Universal Robots PolyScope program: 958_16_OCT_2021_IZQ.urp

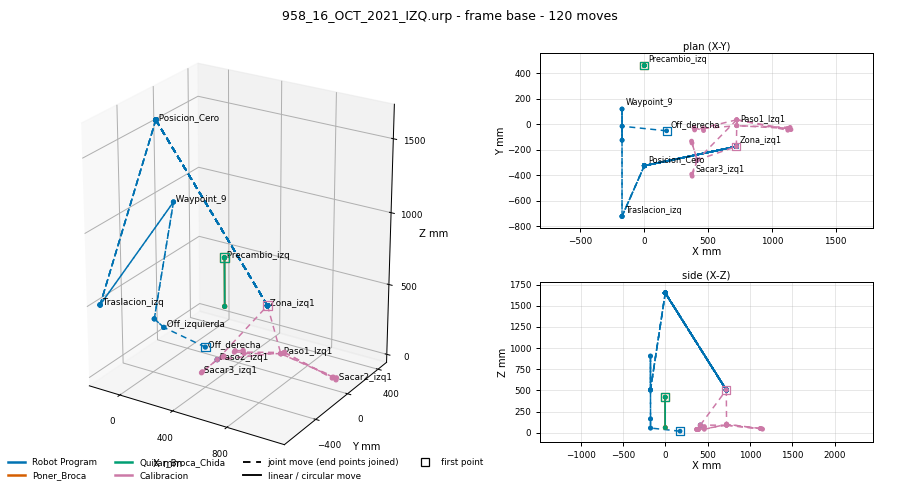
[picture p0: tool path of 958_16_OCT_2021_IZQ.urp in frame base, 120 of 216 moves have a stored position in this frame; points joined in program order, loops and branches not executed]
Program 958_16_OCT_2021_IZQ (installation=instalacion_derecha_10_MAR_21 directory=/programs/FAI3 createdIn=5.6.0.90886 lastSavedIn=5.11.1.108318 robotSerialNumber=20195001785)
Calibrated DH parameters: a=[0.000107, -0.568984, -0.552934, -0.00001, -0.000063, 0]; d=[0.180718, -257.998067, 200.685024, 57.48776, 0.119923, 0.115353]; alpha=[1.571119, 0.000876, -0.002498, 1.571178, -1.570523, 0]; deltaTheta=[0, -0.378191, 0.631587, -0.253396, 0, 0]
Robot Program (runOnlyOnce=false)
  SuppressedNode
    Folder Pruebas_cambiador
      MoveJ speed 60 deg/s, acceleration 80 deg/s^2 (useActiveTCP=true) feature=Base
        Waypoint Precambio_izq: TCP in base x=0.343 y=460.224 z=419.989 mm, rx=0.2109 ry=3.1246 rz=-0.0222 rad; joints [-122.778, -120.749, 120.698, 0.478, 59.722, -0.747] deg; TCP offset x=0.151 y=-167.165 z=35.088 mm, rx=1.5784 ry=-0.0729 rz=0.0687 rad
      Loop Forever
        Call Poner_Broca
        Call Quitar_Broca_Chida
  SuppressedNode
    'Programa'
  Set DigitalOutput pin=salida0; digitalValue=1
  broca := 1645
  Script: textmsg("----------DAS-----------")
  Set ExpressionOutput pin=mensaje_mw10; expression=15
  Wait DigitalInput pin=Continuar_M30; digitalValue=1
  Wait Sleep waitTime=1
  If Lado_Correr≟1
    Folder Arranque
      MoveJ speed 30 deg/s, acceleration 50 deg/s^2 (useActiveTCP=true) feature=Base
        Waypoint Off_derecha: TCP in base x=175.169 y=-51.554 z=18.125 mm, rx=-2.0046 ry=0.0915 rz=0.0578 rad; joints [90.003, -90, 154.529, 0, 89.998, -0.004] deg
        Waypoint Off_izquierda: TCP in base x=-173.642 y=-15.442 z=55.621 mm, rx=-1.8394 ry=0.083 rz=0.0614 rad; joints [-89.997, -89.996, -154.003, -190.002, -89.995, 0.005] deg
      Set DigitalOutput pin=postrnas_m187; digitalValue=1
      Wait Sleep waitTime=1
      Set DigitalOutput pin=Home_M20; digitalValue=1
      Wait Sleep waitTime=1
      Set DigitalOutput pin=postrnas_m187; digitalValue=0
      Set DigitalOutput pin=Home_M20; digitalValue=0
      Set ExpressionOutput pin=mensaje_mw10; expression=20
      Wait DigitalInput pin=Continuar_M30; digitalValue=1
      Wait Sleep waitTime=1
    Folder Traslacion
      Set ExpressionOutput pin=mensaje_mw10; expression=25
      Wait DigitalInput pin=Continuar_M30; digitalValue=1
      Wait Sleep waitTime=1
      MoveJ speed 60 deg/s, acceleration 80 deg/s^2 (useActiveTCP=true) feature=Base
        Waypoint Waypoint_8: TCP in base x=-173.7 y=-124.883 z=163.166 mm, rx=3.1302 ry=-0.1403 rz=0.0027 rad; joints [-90.002, -15, -153.998, -189.998, -89.998, -0.004] deg
        Waypoint Waypoint_9: TCP in base x=-174.329 y=119.284 z=905.669 mm, rx=2.0147 ry=-0.0908 rz=0.0576 rad; joints [-90.002, -15.002, -90.002, -189.996, -89.997, -0.004] deg
        Waypoint Traslacion_izq: TCP in base x=-174.237 y=-721.63 z=505.386 mm, rx=-3.1292 ry=0.1412 rz=-0.0002 rad; joints [-90, -90.001, -90.002, -180, -90.003, -0.001] deg
      Set ExpressionOutput pin=mensaje_mw10; expression=30
      Wait DigitalInput pin=Continuar_M30; digitalValue=1
      Wait Sleep waitTime=1
      Set DigitalOutput pin=postrnas_m187; digitalValue=1
      Wait Sleep waitTime=1
      Set DigitalOutput pin=pos1_izq_m22; digitalValue=1
      Wait Sleep waitTime=2
      Set DigitalOutput pin=pos1_izq_m22; digitalValue=0
      Set DigitalOutput pin=postrnas_m187; digitalValue=0
      Wait Sleep waitTime=5
      Set ExpressionOutput pin=mensaje_mw10; expression=35
      Wait DigitalInput pin=Continuar_M30; digitalValue=1
      Wait Sleep waitTime=1
    Folder Brocas
      Set DigitalOutput pin=carrusel_home; digitalValue=1
      Wait Sleep waitTime=1
      Set DigitalOutput pin=carrusel_home; digitalValue=0
      Set ExpressionOutput pin=mensaje_mw10; expression=40
      Wait DigitalInput pin=Continuar_M30; digitalValue=1
      Wait Sleep waitTime=1
      Set DigitalOutput pin=carrusel_home; digitalValue=1
      Wait Sleep waitTime=1
      Set DigitalOutput pin=carrusel_home; digitalValue=0
      Set ExpressionOutput pin=mensaje_mw10; expression=45
      Wait DigitalInput pin=Continuar_M30; digitalValue=1
      Wait Sleep waitTime=1
      Call Poner_Broca
    Folder Offsets factor
      SuppressedNode
        broca := 1645
      L1B1x := ((0.09523476)/(0.09525))*(0.09523476)
      L1B1y := ((-0.01278382)/(-0.0127))*(-0.01278382)
      L1B2x := ((0.75575414)/(0.75565))*(0.75575414)
      L1B2y := ((-0.01279398)/(-0.0127))*(-0.01279398)
      L2B1x := ((0.09675299)/(0.09525))*(0.09675299)
      L2B1y := ((0.3937)/(0.3937))*(0.3937)
      L2B2x := ((0.757306777)/(0.75565))*(0.757306777)
      L2B2y := ((0.393684081)/(0.3937))*(0.393684081)
    Folder Calibracion
      Set ExpressionOutput pin=mensaje_mw10; expression=50
      Wait DigitalInput pin=Continuar_M30; digitalValue=1
      Wait Sleep waitTime=1
      MoveJ speed 60 deg/s, acceleration 80 deg/s^2 (useActiveTCP=true) feature=Base
        Waypoint Posicion_Cero: TCP in base x=0.551 y=-324.742 z=1651.532 mm, rx=-0.0041 ry=-0.0154 rz=-3.05 rad; joints [-0.003, -90.003, 0.004, -89.999, -0.001, 0] deg
        Waypoint Zona_izq1: TCP in base x=721.637 y=-174.262 z=505.425 mm, rx=2.3235 ry=2.1144 rz=0.0001 rad; joints [0.067, -89.734, -90.405, -179.332, -89.71, -0.034] deg
      broca := 1645
      Set ExpressionOutput pin=mensaje_mw10; expression=125
      Wait DigitalInput pin=Continuar_M30; digitalValue=1
      Wait Sleep waitTime=1
      Set ExpressionOutput pin=mensaje_mw10; expression=130
      Wait DigitalInput pin=Continuar_M30; digitalValue=1
      Wait Sleep waitTime=1
      Call Calibracion
    Folder GoNoGo
      Set ExpressionOutput pin=mensaje_mw10; expression=55
      Wait DigitalInput pin=Continuar_M30; digitalValue=1
      Wait Sleep waitTime=1
      Set ExpressionOutput pin=mensaje_mw10; expression=60
      Wait DigitalInput pin=Continuar_M30; digitalValue=1
      Wait Sleep waitTime=1
      Folder Linea1_Buje1
        Xfin := ((((L1B1x)*(-1)*Xp)-(Xd)-((L1B1y)*(1/m2)))*(-1))*(1)
        Yfin := ((((L1B1y)*(-1)*Yp)-(Yd)+((L1B1x)*(-1)*m1))*(-1))*(1)
        rotaciones := get_actual_tcp_pose()
        var_3 := rotaciones[3]
        var_4 := rotaciones[4]
        var_5 := rotaciones[5]
        If broca≟1645
          PosFinal := p[Xfin-0.00208915,Yfin-0.00208915,0.15,var_3,var_4,var_5]
        ElseIf broca≟1935
          PosFinal := p[Xfin-0.00245745,Yfin-0.00245745,0.15,var_3,var_4,var_5]
        ElseIf broca≟217
          PosFinal := p[Xfin-0.0027559,Yfin-0.0027559,0.15,var_3,var_4,var_5]
        Buje_Final := PosFinal
      MoveJ speed 60 deg/s, acceleration 80 deg/s^2 (useActiveTCP=true) feature=Base
        Waypoint Waypoint (Variable): variable(name=Buje_Final)
      Wait Sleep waitTime=1
      Folder Alturas
        If P1h[2]<P2h[2]
          tcp_chido := get_actual_tcp_pose()
          offset_bajada := p[tcp_chido[0],tcp_chido[1],((alta-0.0095)-(altura/1000)),tcp_chido[3],tcp_chido[4],tcp_chido[5]]
          MoveL speed 15 mm/s, acceleration 30 mm/s^2 (useActiveTCP=true) feature=Base
            Waypoint Waypoint (Variable): variable(name=offset_bajada)
        Else 
          tcp_chido := get_actual_tcp_pose()
          offset_bajada := p[tcp_chido[0],tcp_chido[1],((alta-0.0095)),tcp_chido[3],tcp_chido[4],tcp_chido[5]]
          MoveL speed 15 mm/s, acceleration 30 mm/s^2 (useActiveTCP=true) feature=Base
            Waypoint Waypoint (Variable): variable=offset_bajada
      MoveL speed 15 mm/s, acceleration 30 mm/s^2 (useActiveTCP=true) feature=Base
        Folder Freemove
          Wait Sleep waitTime=2
          Script: freedrive_mode()
          Wait Sleep waitTime=2.5
          Script: end_freedrive_mode()
          var_13 := get_actual_tcp_pose()
          var_13 := p[var_13[0]*1000,var_13[1]*1000,420,420,420,420]
          var_13 := get_actual_tcp_pose()
          var_13 := p[var_13[0],var_13[1],0.1,var_13[3],var_13[4],var_13[5]]
        MoveDirectionNode (selectedDirection=ZPlus)
          Until DISTANCE (allowActions=false deceleration=3 distanceNodeType=STOP) Distance=0.15; motionParameters(blendRadius=0)
      L1B1 := var_13
      Folder Linea1_Buje2
        Xfin := ((((L1B2x)*(-1)*Xp)-(Xd)-((L1B2y)*(1/m2)))*(-1))*(1)
        Yfin := ((((L1B2y)*(-1)*Yp)-(Yd)+((L1B2x)*(-1)*m1))*(-1))*(1)
        rotaciones := get_actual_tcp_pose()
        var_3 := rotaciones[3]
        var_4 := rotaciones[4]
        var_5 := rotaciones[5]
        If broca≟1645
          PosFinal := p[Xfin-0.00208915,Yfin-0.00208915,0.15,var_3,var_4,var_5]
        ElseIf broca≟1935
          PosFinal := p[Xfin-0.00245745,Yfin-0.00245745,0.15,var_3,var_4,var_5]
        ElseIf broca≟217
          PosFinal := p[Xfin-0.0027559,Yfin-0.0027559,0.15,var_3,var_4,var_5]
        Buje_Final := PosFinal
      MoveJ speed 60 deg/s, acceleration 80 deg/s^2 (useActiveTCP=true) feature=Base
        Waypoint Waypoint (Variable): variable=Buje_Final
      Wait Sleep waitTime=1
      Folder Alturas
        If P1h[2]<P2h[2]
          tcp_chido := get_actual_tcp_pose()
          offset_bajada := p[tcp_chido[0],tcp_chido[1],((alta-0.0095)),tcp_chido[3],tcp_chido[4],tcp_chido[5]]
          MoveL speed 15 mm/s, acceleration 30 mm/s^2 (useActiveTCP=true) feature=Base
            Waypoint Waypoint (Variable): variable=offset_bajada
        Else 
          tcp_chido := get_actual_tcp_pose()
          offset_bajada := p[tcp_chido[0],tcp_chido[1],((alta-0.0095)-(altura/1000)),tcp_chido[3],tcp_chido[4],tcp_chido[5]]
          MoveL speed 15 mm/s, acceleration 30 mm/s^2 (useActiveTCP=true) feature=Base
            Waypoint Waypoint (Variable): variable=offset_bajada
      MoveL speed 15 mm/s, acceleration 30 mm/s^2 (useActiveTCP=true) feature=Base
        Folder Freemove
          Wait Sleep waitTime=2
          Script: freedrive_mode()
          Wait Sleep waitTime=2.5
          Script: end_freedrive_mode()
          var_13 := get_actual_tcp_pose()
          var_13 := p[var_13[0]*1000,var_13[1]*1000,420,420,420,420]
          var_13 := get_actual_tcp_pose()
          var_13 := p[var_13[0],var_13[1],0.1,var_13[3],var_13[4],var_13[5]]
        MoveDirectionNode (selectedDirection=ZPlus)
          Until DISTANCE (allowActions=false deceleration=3 distanceNodeType=STOP) Distance=0.15; motionParameters(blendRadius=0)
      L1B2 := var_13
      Folder Linea2_Buje2
        Xfin := ((((L2B2x)*(-1)*Xp)-(Xd)-(L2B2y*(1/m2)))*(-1))*(1)
        Yfin := ((((L2B2y)*(-1)*Yp)-(Yd)+((L2B2x)*(-1)*m1))*(-1))*(1)
        rotaciones := get_actual_tcp_pose()
        var_3 := rotaciones[3]
        var_4 := rotaciones[4]
        var_5 := rotaciones[5]
        If broca≟1645
          PosFinal := p[Xfin-0.00208915,Yfin-0.00208915,0.15,var_3,var_4,var_5]
        ElseIf broca≟1935
          PosFinal := p[Xfin-0.00245745,Yfin-0.00245745,0.15,var_3,var_4,var_5]
        ElseIf broca≟217
          PosFinal := p[Xfin-0.0027559,Yfin-0.0027559,0.15,var_3,var_4,var_5]
        Buje_Final := PosFinal
      MoveJ speed 60 deg/s, acceleration 80 deg/s^2 (useActiveTCP=true) feature=Base
        Waypoint Waypoint (Variable): variable=Buje_Final
      Wait Sleep waitTime=1
      Folder Alturas
        If P1h[2]<P2h[2]
          tcp_chido := get_actual_tcp_pose()
          offset_bajada := p[tcp_chido[0],tcp_chido[1],((alta-0.0095)),tcp_chido[3],tcp_chido[4],tcp_chido[5]]
          MoveL speed 15 mm/s, acceleration 30 mm/s^2 (useActiveTCP=true) feature=Base
            Waypoint Waypoint (Variable): variable=offset_bajada
        Else 
          tcp_chido := get_actual_tcp_pose()
          offset_bajada := p[tcp_chido[0],tcp_chido[1],((alta-0.0095)-(altura/1000)),tcp_chido[3],tcp_chido[4],tcp_chido[5]]
          MoveL speed 15 mm/s, acceleration 30 mm/s^2 (useActiveTCP=true) feature=Base
            Waypoint Waypoint (Variable): variable=offset_bajada
      MoveL speed 15 mm/s, acceleration 30 mm/s^2 (useActiveTCP=true) feature=Base
        Folder Freemove
          Wait Sleep waitTime=2
          Script: freedrive_mode()
          Wait Sleep waitTime=2.5
          Script: end_freedrive_mode()
          var_13 := get_actual_tcp_pose()
          var_13 := p[var_13[0]*1000,var_13[1]*1000,420,420,420,420]
          var_13 := get_actual_tcp_pose()
          var_13 := p[var_13[0],var_13[1],0.1,var_13[3],var_13[4],var_13[5]]
        MoveDirectionNode (selectedDirection=ZPlus)
          Until DISTANCE (allowActions=false deceleration=3 distanceNodeType=STOP) Distance=0.15; motionParameters(blendRadius=0)
      L2B2 := var_13
      Folder Linea2_Buje1
        Xfin := ((((L2B1x)*(-1)*Xp)-(Xd)-((L2B1y)*(1/m2)))*(-1))*(1)
        Yfin := ((((L2B1y)*(-1)*Yp)-(Yd)+((L2B1x)*(-1)*m1))*(-1))*(1)
        rotaciones := get_actual_tcp_pose()
        var_3 := rotaciones[3]
        var_4 := rotaciones[4]
        var_5 := rotaciones[5]
        If broca≟1645
          PosFinal := p[Xfin-0.00208915,Yfin-0.00208915,0.15,var_3,var_4,var_5]
        ElseIf broca≟1935
          PosFinal := p[Xfin-0.00245745,Yfin-0.00245745,0.15,var_3,var_4,var_5]
        ElseIf broca≟217
          PosFinal := p[Xfin-0.0027559,Yfin-0.0027559,0.15,var_3,var_4,var_5]
        Buje_Final := PosFinal
      MoveJ speed 60 deg/s, acceleration 80 deg/s^2 (useActiveTCP=true) feature=Base
        Waypoint Paso2_izq1: TCP in base x=414.118 y=-280.673 z=89.978 mm, rx=-2.3928 ry=-2.0356 rz=0 rad; joints [-18.236, -84.335, -142.099, -133.065, -104.295, 0.11] deg
        Waypoint Waypoint (Variable): variable=Buje_Final
      Wait Sleep waitTime=1
      Folder Alturas
        If P1h[2]<P2h[2]
          tcp_chido := get_actual_tcp_pose()
          offset_bajada := p[tcp_chido[0],tcp_chido[1],((alta-0.0095)-(altura/1000)),tcp_chido[3],tcp_chido[4],tcp_chido[5]]
          MoveL speed 15 mm/s, acceleration 30 mm/s^2 (useActiveTCP=true) feature=Base
            Waypoint Waypoint (Variable): variable=offset_bajada
        Else 
          tcp_chido := get_actual_tcp_pose()
          offset_bajada := p[tcp_chido[0],tcp_chido[1],((alta-0.0095)),tcp_chido[3],tcp_chido[4],tcp_chido[5]]
          MoveL speed 15 mm/s, acceleration 30 mm/s^2 (useActiveTCP=true) feature=Base
            Waypoint Waypoint (Variable): variable=offset_bajada
      MoveL speed 15 mm/s, acceleration 30 mm/s^2 (useActiveTCP=true) feature=Base
        Folder Freemove
          Wait Sleep waitTime=2
          Script: freedrive_mode()
          Wait Sleep waitTime=2.5
          Script: end_freedrive_mode()
          var_13 := get_actual_tcp_pose()
          var_13 := p[var_13[0]*1000,var_13[1]*1000,420,420,420,420]
          var_13 := get_actual_tcp_pose()
          var_13 := p[var_13[0],var_13[1],0.1,var_13[3],var_13[4],var_13[5]]
        MoveDirectionNode (selectedDirection=ZPlus)
          Until DISTANCE (allowActions=false deceleration=3 distanceNodeType=STOP) Distance=0.15; motionParameters(blendRadius=0)
      MoveJ speed 60 deg/s, acceleration 80 deg/s^2 (useActiveTCP=true) feature=Base
        Waypoint Zona_izq1: TCP in base x=721.637 y=-174.262 z=505.425 mm, rx=2.3235 ry=2.1144 rz=0.0001 rad; joints [0.067, -89.734, -90.405, -179.332, -89.71, -0.034] deg
      L2B1 := var_13
    SuppressedNode
      Folder Cancelar barrenado
        MoveJ speed 60 deg/s, acceleration 80 deg/s^2 (useActiveTCP=true) feature=Base
          SuppressedNode
            Waypoint Zona_der1: TCP in base x=-724.618 y=-175.006 z=455.096 mm, rx=2.0346 ry=-2.3862 rz=-0.0105 rad; joints [0.001, -89.997, 90, 0.002, 90.001, 0.002] deg; TCP offset x=0.411 y=-218.298 z=37.994 mm, rx=1.558 ry=-0.1255 rz=0.1212 rad
          Waypoint Zona_izq1: TCP in base x=721.637 y=-174.262 z=505.425 mm, rx=2.3235 ry=2.1144 rz=0.0001 rad; joints [0.067, -89.734, -90.405, -179.332, -89.71, -0.034] deg; TCP offset x=0.151 y=-167.165 z=35.088 mm, rx=1.5784 ry=-0.0729 rz=0.0687 rad
          Waypoint Posicion_Cero: TCP in base x=0.551 y=-324.742 z=1651.532 mm, rx=-0.0041 ry=-0.0154 rz=-3.05 rad; joints [-0.003, -90.003, 0.004, -89.999, -0.001, 0] deg
        Call Quitar_Broca_Chida
        Set ExpressionOutput pin=mensaje_mw10; expression=100
        Wait DigitalInput pin=Continuar_M30; digitalValue=1
        Wait Sleep waitTime=1
        Set ExpressionOutput pin=mensaje_mw10; expression=155
        Wait DigitalInput pin=Continuar_M30; digitalValue=1
        Wait Sleep waitTime=1
    Folder Colocar broca
      Call Quitar_Broca_Chida
      Call Poner_Broca
    Folder Barrenado1
      Set ExpressionOutput pin=mensaje_mw10; expression=65
      Wait DigitalInput pin=Continuar_M30; digitalValue=1
      Wait Sleep waitTime=1
      Set ExpressionOutput pin=mensaje_mw10; expression=150
      Wait Sleep waitTime=1
      Folder Linea 1 a 1645
        broca := 1645
        Folder Buje_inicial
          Buje_Inicial := L1B2
        Folder Buje_final
          Buje_Final := L1B1
        barrenosTotales := 27
        barrenoActual := 1
        Loop While (checkContinuously=false) expression=barrenoActual≤barrenosTotales
          MoveL speed 250 mm/s, acceleration 1200 mm/s^2 (useActiveTCP=true) feature=Base
            bajada_broca := p[0,0,0.006,0,0,0]
            internos := interpolate_pose(Buje_Inicial, Buje_Final, ((barrenoActual)-1)/((barrenosTotales)-1))
            Folder Alturas
              If barrenoActual≟3 or barrenoActual≟5 or barrenoActual≟7 or barrenoActual≟9 or barrenoActual≟11 or barrenoActual≟13 or barrenoActual≟15 or barrenoActual≟17 or barrenoActual≟19 or barrenoActual≟21 or barrenoActual≟23 or barrenoActual≟25 or barrenoActual≟27 or barrenoActual≟1
                Set ExpressionOutput pin=mensaje_mw10; expression=200
                Wait DigitalInput pin=Continuar_M30; digitalValue=1
                Wait Sleep waitTime=1
                Set ExpressionOutput pin=mensaje_mw10; expression=150
                Wait Sleep waitTime=1
              MoveJ speed 60 deg/s, acceleration 80 deg/s^2 (useActiveTCP=true) feature=Base
                Waypoint Waypoint (Variable): variable(name=internos)
              Wait Sleep waitTime=2
              If P1h[2]<P2h[2]
                acomodin := (altura/(barrenosTotales-1))*(barrenoActual-1)
                tcp_chido := get_actual_tcp_pose()
                offset_bajada := p[tcp_chido[0],tcp_chido[1],((alta-0.0095)-(acomodin/1000)),tcp_chido[3],tcp_chido[4],tcp_chido[5]]
                MoveL speed 15 mm/s, acceleration 30 mm/s^2 (useActiveTCP=true) feature=Base
                  Waypoint Waypoint (Variable): variable=offset_bajada
              Else 
                acomodin := (altura/(barrenosTotales-1))*(26-(barrenoActual-1))
                tcp_chido := get_actual_tcp_pose()
                offset_bajada := p[tcp_chido[0],tcp_chido[1],((alta-0.0095)-(acomodin/1000)),tcp_chido[3],tcp_chido[4],tcp_chido[5]]
                MoveL speed 15 mm/s, acceleration 30 mm/s^2 (useActiveTCP=true) feature=Base
                  Waypoint Waypoint (Variable): variable=offset_bajada
            Folder Freemove
              Wait Sleep waitTime=2
              Script: freedrive_mode()
              Wait Sleep waitTime=2.5
              Script: end_freedrive_mode()
            Wait Sleep waitTime=0.3
            Set DigitalOutput pin=config_out[1]; digitalValue=1
            Wait Sleep waitTime=1
            Wait Sleep waitTime=0.3
            Wait Sleep waitTime=0.3
            Wait Sleep waitTime=0.3
            Loop Counting (count=3) loopVariable(name=Loop_4)
              Poses_taladrado := pose_sub(get_actual_tcp_pose(), bajada_broca)
              Waypoint Waypoint (Variable): motionParameters(jointSpeed=1.047198 jointAcceleration=1.396263 cartesianSpeed=0.001 cartesianAcceleration=0.005); variable(name=Poses_taladrado)
              If bajada_broca≟p[0,0,0.018,0,0,0]
                num_barreno := str_cat("Barreno: ",barrenoActual)
                tcp_actual := get_actual_tcp_pose()
                X_actual := str_cat("     X: ",tcp_actual[0])
                Y_actual := str_cat("     Y: ",tcp_actual[1])
                pos_barreno := str_cat(X_actual,Y_actual)
                Script: textmsg(num_barreno,pos_barreno)
              Poses_taladrado := pose_add(get_actual_tcp_pose(), bajada_broca)
              Waypoint Waypoint (Variable): motionParameters(jointSpeed=1.047198 jointAcceleration=1.396263 cartesianSpeed=0.01 cartesianAcceleration=0.01); variable=Poses_taladrado
              bajada_broca := pose_add(bajada_broca, p[0,0,0.006,0,0,0])
            MoveDirectionNode (selectedDirection=ZPlus toolParams=0.03, 0.04)
              Until DISTANCE (allowActions=false deceleration=3 distanceNodeType=STOP) Distance=0.05; motionParameters(blendRadius=0)
            MoveJ speed 60 deg/s, acceleration 80 deg/s^2 (useActiveTCP=true) feature=Base
              Waypoint Waypoint (Variable): variable=internos
            Wait Sleep waitTime=0.3
            Set DigitalOutput pin=config_out[1]; digitalValue=0
            Wait Sleep waitTime=0.3
            If barrenoActual≟13 or barrenoActual≟27
              MoveDirectionNode (selectedDirection=ZPlus toolParams=0.03, 0.04)
                Until DISTANCE (allowActions=false deceleration=3 distanceNodeType=STOP) Distance=0.03; motionParameters(blendRadius=0)
              MoveJ speed 60 deg/s, acceleration 80 deg/s^2 (useActiveTCP=true) feature=Base
                Waypoint Zona_izq1: TCP in base x=721.637 y=-174.262 z=505.425 mm, rx=2.3235 ry=2.1144 rz=0.0001 rad; joints [0.067, -89.734, -90.405, -179.332, -89.71, -0.034] deg
                Waypoint Posicion_Cero: TCP in base x=0.551 y=-324.742 z=1651.532 mm, rx=-0.0041 ry=-0.0154 rz=-3.05 rad; joints [-0.003, -90.003, 0.004, -89.999, -0.001, 0] deg
              Call Quitar_Broca_Chida
              Call Poner_Broca
              MoveJ speed 60 deg/s, acceleration 80 deg/s^2 (useActiveTCP=true) feature=Base
                Waypoint Posicion_Cero: TCP in base x=0.551 y=-324.742 z=1651.532 mm, rx=-0.0041 ry=-0.0154 rz=-3.05 rad; joints [-0.003, -90.003, 0.004, -89.999, -0.001, 0] deg
                Waypoint Zona_izq1: TCP in base x=721.637 y=-174.262 z=505.425 mm, rx=2.3235 ry=2.1144 rz=0.0001 rad; joints [0.067, -89.734, -90.405, -179.332, -89.71, -0.034] deg
            barrenoActual := barrenoActual+1
      Folder Linea 2 a 1645
        broca := 1645
        Folder Buje_inicial
          Buje_Inicial := L2B2
        Folder Buje_final
          Buje_Final := L2B1
        barrenosTotales := 27
        barrenoActual := 1
        Loop While (checkContinuously=false) expression=barrenoActual≤barrenosTotales
          MoveL speed 250 mm/s, acceleration 1200 mm/s^2 (useActiveTCP=true) feature=Base
            bajada_broca := p[0,0,0.006,0,0,0]
            internos := interpolate_pose(Buje_Inicial, Buje_Final, ((barrenoActual)-1)/((barrenosTotales)-1))
            Folder Alturas
              If barrenoActual≟3 or barrenoActual≟5 or barrenoActual≟7 or barrenoActual≟9 or barrenoActual≟11 or barrenoActual≟13 or barrenoActual≟15 or barrenoActual≟17 or barrenoActual≟19 or barrenoActual≟21 or barrenoActual≟23 or barrenoActual≟25 or barrenoActual≟27 or barrenoActual≟1
                Set ExpressionOutput pin=mensaje_mw10; expression=200
                Wait DigitalInput pin=Continuar_M30; digitalValue=1
                Wait Sleep waitTime=1
                Set ExpressionOutput pin=mensaje_mw10; expression=150
                Wait Sleep waitTime=1
              MoveJ speed 60 deg/s, acceleration 80 deg/s^2 (useActiveTCP=true) feature=Base
                Waypoint Waypoint (Variable): variable=internos
              Wait Sleep waitTime=2
              If P1h[2]<P2h[2]
                acomodin := (altura/(barrenosTotales-1))*(barrenoActual-1)
                tcp_chido := get_actual_tcp_pose()
                offset_bajada := p[tcp_chido[0],tcp_chido[1],((alta-0.0095)-(acomodin/1000)),tcp_chido[3],tcp_chido[4],tcp_chido[5]]
                MoveL speed 15 mm/s, acceleration 30 mm/s^2 (useActiveTCP=true) feature=Base
                  Waypoint Waypoint (Variable): variable=offset_bajada
              Else 
                acomodin := (altura/(barrenosTotales-1))*(26-(barrenoActual-1))
                tcp_chido := get_actual_tcp_pose()
                offset_bajada := p[tcp_chido[0],tcp_chido[1],((alta-0.0095)-(acomodin/1000)),tcp_chido[3],tcp_chido[4],tcp_chido[5]]
                MoveL speed 15 mm/s, acceleration 30 mm/s^2 (useActiveTCP=true) feature=Base
                  Waypoint Waypoint (Variable): variable=offset_bajada
            Folder Freemove
              Wait Sleep waitTime=2
              Script: freedrive_mode()
              Wait Sleep waitTime=2.5
              Script: end_freedrive_mode()
            Wait Sleep waitTime=0.3
            Set DigitalOutput pin=config_out[1]; digitalValue=1
            Wait Sleep waitTime=1
            Wait Sleep waitTime=0.3
            Wait Sleep waitTime=0.3
            Wait Sleep waitTime=0.3
            Loop Counting (count=3) loopVariable(name=Loop_12)
              Poses_taladrado := pose_sub(get_actual_tcp_pose(), bajada_broca)
              Waypoint Waypoint (Variable): motionParameters(jointSpeed=1.047198 jointAcceleration=1.396263 cartesianSpeed=0.001 cartesianAcceleration=0.005); variable=Poses_taladrado
              If bajada_broca≟p[0,0,0.018,0,0,0]
                num_barreno := str_cat("Barreno: ",barrenoActual)
                tcp_actual := get_actual_tcp_pose()
                X_actual := str_cat("     X: ",tcp_actual[0])
                Y_actual := str_cat("     Y: ",tcp_actual[1])
                pos_barreno := str_cat(X_actual,Y_actual)
                Script: textmsg(num_barreno,pos_barreno)
              Poses_taladrado := pose_add(get_actual_tcp_pose(), bajada_broca)
              Waypoint Waypoint (Variable): motionParameters(jointSpeed=1.047198 jointAcceleration=1.396263 cartesianSpeed=0.01 cartesianAcceleration=0.01); variable=Poses_taladrado
              bajada_broca := pose_add(bajada_broca, p[0,0,0.006,0,0,0])
            MoveDirectionNode (selectedDirection=ZPlus toolParams=0.03, 0.04)
              Until DISTANCE (allowActions=false deceleration=3 distanceNodeType=STOP) Distance=0.05; motionParameters(blendRadius=0)
            MoveJ speed 60 deg/s, acceleration 80 deg/s^2 (useActiveTCP=true) feature=Base
              Waypoint Waypoint (Variable): variable=internos
            Wait Sleep waitTime=0.3
            Set DigitalOutput pin=config_out[1]; digitalValue=0
            Wait Sleep waitTime=0.3
            If barrenoActual≟13
              MoveDirectionNode (selectedDirection=ZPlus)
                Until DISTANCE (allowActions=false deceleration=3 distanceNodeType=STOP) Distance=0.03; motionParameters(blendRadius=0)
              MoveJ speed 60 deg/s, acceleration 80 deg/s^2 (useActiveTCP=true) feature=Base
                Waypoint Zona_izq1: TCP in base x=721.637 y=-174.262 z=505.425 mm, rx=2.3235 ry=2.1144 rz=0.0001 rad; joints [0.067, -89.734, -90.405, -179.332, -89.71, -0.034] deg
                Waypoint Posicion_Cero: TCP in base x=0.551 y=-324.742 z=1651.532 mm, rx=-0.0041 ry=-0.0154 rz=-3.05 rad; joints [-0.003, -90.003, 0.004, -89.999, -0.001, 0] deg
              Call Quitar_Broca_Chida
              Call Poner_Broca
              MoveJ speed 60 deg/s, acceleration 80 deg/s^2 (useActiveTCP=true) feature=Base
                Waypoint Posicion_Cero: TCP in base x=0.551 y=-324.742 z=1651.532 mm, rx=-0.0041 ry=-0.0154 rz=-3.05 rad; joints [-0.003, -90.003, 0.004, -89.999, -0.001, 0] deg
                Waypoint Zona_izq1: TCP in base x=721.637 y=-174.262 z=505.425 mm, rx=2.3235 ry=2.1144 rz=0.0001 rad; joints [0.067, -89.734, -90.405, -179.332, -89.71, -0.034] deg
            ElseIf barrenoActual≟27
              MoveDirectionNode (selectedDirection=ZPlus)
                Until DISTANCE (allowActions=false deceleration=3 distanceNodeType=STOP) Distance=0.03; motionParameters(blendRadius=0)
              MoveJ speed 60 deg/s, acceleration 80 deg/s^2 (useActiveTCP=true) feature=Base
                Waypoint Zona_izq1: TCP in base x=721.637 y=-174.262 z=505.425 mm, rx=2.3235 ry=2.1144 rz=0.0001 rad; joints [0.067, -89.734, -90.405, -179.332, -89.71, -0.034] deg
                Waypoint Posicion_Cero: TCP in base x=0.551 y=-324.742 z=1651.532 mm, rx=-0.0041 ry=-0.0154 rz=-3.05 rad; joints [-0.003, -90.003, 0.004, -89.999, -0.001, 0] deg
              Call Quitar_Broca_Chida
              Set DigitalOutput pin=carrusel_home; digitalValue=1
              Wait Sleep waitTime=1
              Set DigitalOutput pin=carrusel_home; digitalValue=0
              Set ExpressionOutput pin=mensaje_mw10; expression=70
              Wait DigitalInput pin=Continuar_M30; digitalValue=1
              Wait Sleep waitTime=1
              Set ExpressionOutput pin=mensaje_mw10; expression=120
              Wait DigitalInput pin=Continuar_M30; digitalValue=1
              Wait Sleep waitTime=1
              Set DigitalOutput pin=carrusel_home; digitalValue=1
              Wait Sleep waitTime=1
              Set DigitalOutput pin=carrusel_home; digitalValue=0
              Set ExpressionOutput pin=mensaje_mw10; expression=75
              Wait DigitalInput pin=Continuar_M30; digitalValue=1
              Wait Sleep waitTime=1
              Call Poner_Broca
              broca := 1935
              MoveJ speed 60 deg/s, acceleration 80 deg/s^2 (useActiveTCP=true) feature=Base
                Waypoint Posicion_Cero: TCP in base x=0.551 y=-324.742 z=1651.532 mm, rx=-0.0041 ry=-0.0154 rz=-3.05 rad; joints [-0.003, -90.003, 0.004, -89.999, -0.001, 0] deg
                Waypoint Zona_izq1: TCP in base x=721.637 y=-174.262 z=505.425 mm, rx=2.3235 ry=2.1144 rz=0.0001 rad; joints [0.067, -89.734, -90.405, -179.332, -89.71, -0.034] deg
              Set ExpressionOutput pin=mensaje_mw10; expression=80
              Wait DigitalInput pin=Continuar_M30; digitalValue=1
              Wait Sleep waitTime=1
              Set ExpressionOutput pin=mensaje_mw10; expression=150
              Wait DigitalInput pin=Continuar_M30; digitalValue=1
              Wait Sleep waitTime=1
            barrenoActual := barrenoActual+1
      Folder Linea 1 a 1935
        broca := 1935
        Folder Buje_inicial
          Buje_Inicial := L1B2
        Folder Buje_final
          Buje_Final := L1B1
        barrenosTotales := 27
        barrenoActual := 1
        Loop While (checkContinuously=false) expression=barrenoActual≤barrenosTotales
          MoveL speed 250 mm/s, acceleration 1200 mm/s^2 (useActiveTCP=true) feature=Base
            bajada_broca := p[0,0,0.009,0,0,0]
            internos := interpolate_pose(Buje_Inicial, Buje_Final, ((barrenoActual)-1)/((barrenosTotales)-1))
            Folder Alturas
              If barrenoActual≟3 or barrenoActual≟5 or barrenoActual≟7 or barrenoActual≟9 or barrenoActual≟11 or barrenoActual≟13 or barrenoActual≟15 or barrenoActual≟17 or barrenoActual≟19 or barrenoActual≟21 or barrenoActual≟23 or barrenoActual≟25 or barrenoActual≟27 or barrenoActual≟1
                Set ExpressionOutput pin=mensaje_mw10; expression=200
                Wait DigitalInput pin=Continuar_M30; digitalValue=1
                Wait Sleep waitTime=1
                Set ExpressionOutput pin=mensaje_mw10; expression=150
                Wait Sleep waitTime=1
              MoveJ speed 60 deg/s, acceleration 80 deg/s^2 (useActiveTCP=true) feature=Base
                Waypoint Waypoint (Variable): variable=internos
              Wait Sleep waitTime=2
              If P1h[2]<P2h[2]
                acomodin := (altura/(barrenosTotales-1))*(barrenoActual-1)
                tcp_chido := get_actual_tcp_pose()
                offset_bajada := p[tcp_chido[0],tcp_chido[1],((alta-0.0095)-(acomodin/1000)),tcp_chido[3],tcp_chido[4],tcp_chido[5]]
                MoveL speed 15 mm/s, acceleration 30 mm/s^2 (useActiveTCP=true) feature=Base
                  Waypoint Waypoint (Variable): variable=offset_bajada
              Else 
                acomodin := (altura/(barrenosTotales-1))*(26-(barrenoActual-1))
                tcp_chido := get_actual_tcp_pose()
                offset_bajada := p[tcp_chido[0],tcp_chido[1],((alta-0.0095)-(acomodin/1000)),tcp_chido[3],tcp_chido[4],tcp_chido[5]]
                MoveL speed 15 mm/s, acceleration 30 mm/s^2 (useActiveTCP=true) feature=Base
                  Waypoint Waypoint (Variable): variable=offset_bajada
            Folder Freemove
              Wait Sleep waitTime=2
              Script: freedrive_mode()
              Wait Sleep waitTime=2.5
              Script: end_freedrive_mode()
            Wait Sleep waitTime=0.3
            Set DigitalOutput pin=config_out[1]; digitalValue=1
            Wait Sleep waitTime=1
            Wait Sleep waitTime=0.3
            Wait Sleep waitTime=0.3
            Wait Sleep waitTime=0.3
            Loop Counting (count=2) loopVariable(name=Loop_15)
              Poses_taladrado := pose_sub(get_actual_tcp_pose(), bajada_broca)
              Waypoint Waypoint (Variable): motionParameters(jointSpeed=1.047198 jointAcceleration=1.396263 cartesianSpeed=0.001 cartesianAcceleration=0.005); variable=Poses_taladrado
              If bajada_broca≟p[0,0,0.018,0,0,0]
                num_barreno := str_cat("Barreno: ",barrenoActual)
                tcp_actual := get_actual_tcp_pose()
                X_actual := str_cat("     X: ",tcp_actual[0])
                Y_actual := str_cat("     Y: ",tcp_actual[1])
                pos_barreno := str_cat(X_actual,Y_actual)
                Script: textmsg(num_barreno,pos_barreno)
              Poses_taladrado := pose_add(get_actual_tcp_pose(), bajada_broca)
              Waypoint Waypoint (Variable): motionParameters(jointSpeed=1.047198 jointAcceleration=1.396263 cartesianSpeed=0.01 cartesianAcceleration=0.01); variable=Poses_taladrado
              bajada_broca := pose_add(bajada_broca, p[0,0,0.009,0,0,0])
            MoveDirectionNode (selectedDirection=ZPlus toolParams=0.03, 0.04)
              Until DISTANCE (allowActions=false deceleration=3 distanceNodeType=STOP) Distance=0.05; motionParameters(blendRadius=0)
            MoveJ speed 60 deg/s, acceleration 80 deg/s^2 (useActiveTCP=true) feature=Base
              Waypoint Waypoint (Variable): variable=internos
            Wait Sleep waitTime=0.3
            Set DigitalOutput pin=config_out[1]; digitalValue=0
            Wait Sleep waitTime=0.3
            If barrenoActual≟13 or barrenoActual≟27
              MoveDirectionNode (selectedDirection=ZPlus)
                Until DISTANCE (allowActions=false deceleration=3 distanceNodeType=STOP) Distance=0.03; motionParameters(blendRadius=0)
              MoveJ speed 60 deg/s, acceleration 80 deg/s^2 (useActiveTCP=true) feature=Base
                Waypoint Zona_izq1: TCP in base x=721.637 y=-174.262 z=505.425 mm, rx=2.3235 ry=2.1144 rz=0.0001 rad; joints [0.067, -89.734, -90.405, -179.332, -89.71, -0.034] deg
                Waypoint Posicion_Cero: TCP in base x=0.551 y=-324.742 z=1651.532 mm, rx=-0.0041 ry=-0.0154 rz=-3.05 rad; joints [-0.003, -90.003, 0.004, -89.999, -0.001, 0] deg
              Call Quitar_Broca_Chida
              Call Poner_Broca
              MoveJ speed 60 deg/s, acceleration 80 deg/s^2 (useActiveTCP=true) feature=Base
                Waypoint Posicion_Cero: TCP in base x=0.551 y=-324.742 z=1651.532 mm, rx=-0.0041 ry=-0.0154 rz=-3.05 rad; joints [-0.003, -90.003, 0.004, -89.999, -0.001, 0] deg
                Waypoint Zona_izq1: TCP in base x=721.637 y=-174.262 z=505.425 mm, rx=2.3235 ry=2.1144 rz=0.0001 rad; joints [0.067, -89.734, -90.405, -179.332, -89.71, -0.034] deg
            barrenoActual := barrenoActual+1
      Folder Linea 2 a 1935
        broca := 1935
        Folder Buje_inicial
          Buje_Inicial := L2B2
        Folder Buje_final
          Buje_Final := L2B1
        barrenosTotales := 27
        barrenoActual := 1
        Loop While (checkContinuously=false) expression=barrenoActual≤barrenosTotales
          MoveL speed 250 mm/s, acceleration 1200 mm/s^2 (useActiveTCP=true) feature=Base
            bajada_broca := p[0,0,0.009,0,0,0]
            internos := interpolate_pose(Buje_Inicial, Buje_Final, ((barrenoActual)-1)/((barrenosTotales)-1))
            Folder Alturas
              If barrenoActual≟3 or barrenoActual≟5 or barrenoActual≟7 or barrenoActual≟9 or barrenoActual≟11 or barrenoActual≟13 or barrenoActual≟15 or barrenoActual≟17 or barrenoActual≟19 or barrenoActual≟21 or barrenoActual≟23 or barrenoActual≟25 or barrenoActual≟27 or barrenoActual≟1
                Set ExpressionOutput pin=mensaje_mw10; expression=200
                Wait DigitalInput pin=Continuar_M30; digitalValue=1
                Wait Sleep waitTime=1
                Set ExpressionOutput pin=mensaje_mw10; expression=150
                Wait Sleep waitTime=1
              MoveJ speed 60 deg/s, acceleration 80 deg/s^2 (useActiveTCP=true) feature=Base
                Waypoint Waypoint (Variable): variable=internos
              Wait Sleep waitTime=2
              If P1h[2]<P2h[2]
                acomodin := (altura/(barrenosTotales-1))*(barrenoActual-1)
                tcp_chido := get_actual_tcp_pose()
                offset_bajada := p[tcp_chido[0],tcp_chido[1],((alta-0.0095)-(acomodin/1000)),tcp_chido[3],tcp_chido[4],tcp_chido[5]]
                MoveL speed 15 mm/s, acceleration 30 mm/s^2 (useActiveTCP=true) feature=Base
                  Waypoint Waypoint (Variable): variable=offset_bajada
              Else 
                acomodin := (altura/(barrenosTotales-1))*(26-(barrenoActual-1))
                tcp_chido := get_actual_tcp_pose()
                offset_bajada := p[tcp_chido[0],tcp_chido[1],((alta-0.0095)-(acomodin/1000)),tcp_chido[3],tcp_chido[4],tcp_chido[5]]
                MoveL speed 15 mm/s, acceleration 30 mm/s^2 (useActiveTCP=true) feature=Base
                  Waypoint Waypoint (Variable): variable=offset_bajada
            Folder Freemove
              Wait Sleep waitTime=2
              Script: freedrive_mode()
              Wait Sleep waitTime=2.5
              Script: end_freedrive_mode()
            Wait Sleep waitTime=0.3
            Set DigitalOutput pin=config_out[1]; digitalValue=1
            Wait Sleep waitTime=1
            Wait Sleep waitTime=0.3
            Wait Sleep waitTime=0.3
            Wait Sleep waitTime=0.3
            Loop Counting (count=2) loopVariable(name=Loop_17)
              Poses_taladrado := pose_sub(get_actual_tcp_pose(), bajada_broca)
              Waypoint Waypoint (Variable): motionParameters(jointSpeed=1.047198 jointAcceleration=1.396263 cartesianSpeed=0.001 cartesianAcceleration=0.005); variable=Poses_taladrado
              If bajada_broca≟p[0,0,0.018,0,0,0]
                num_barreno := str_cat("Barreno: ",barrenoActual)
                tcp_actual := get_actual_tcp_pose()
                X_actual := str_cat("     X: ",tcp_actual[0])
                Y_actual := str_cat("     Y: ",tcp_actual[1])
                pos_barreno := str_cat(X_actual,Y_actual)
                Script: textmsg(num_barreno,pos_barreno)
              Poses_taladrado := pose_add(get_actual_tcp_pose(), bajada_broca)
              Waypoint Waypoint (Variable): motionParameters(jointSpeed=1.047198 jointAcceleration=1.396263 cartesianSpeed=0.01 cartesianAcceleration=0.01); variable=Poses_taladrado
              bajada_broca := pose_add(bajada_broca, p[0,0,0.009,0,0,0])
            MoveDirectionNode (selectedDirection=ZPlus toolParams=0.03, 0.04)
              Until DISTANCE (allowActions=false deceleration=3 distanceNodeType=STOP) Distance=0.05; motionParameters(blendRadius=0)
            MoveJ speed 60 deg/s, acceleration 80 deg/s^2 (useActiveTCP=true) feature=Base
              Waypoint Waypoint (Variable): variable=internos
            Wait Sleep waitTime=0.3
            Set DigitalOutput pin=config_out[1]; digitalValue=0
            Wait Sleep waitTime=0.3
            If barrenoActual≟13
              MoveDirectionNode (selectedDirection=ZPlus)
                Until DISTANCE (allowActions=false deceleration=3 distanceNodeType=STOP) Distance=0.03; motionParameters(blendRadius=0)
              MoveJ speed 60 deg/s, acceleration 80 deg/s^2 (useActiveTCP=true) feature=Base
                Waypoint Zona_izq1: TCP in base x=721.637 y=-174.262 z=505.425 mm, rx=2.3235 ry=2.1144 rz=0.0001 rad; joints [0.067, -89.734, -90.405, -179.332, -89.71, -0.034] deg
                Waypoint Posicion_Cero: TCP in base x=0.551 y=-324.742 z=1651.532 mm, rx=-0.0041 ry=-0.0154 rz=-3.05 rad; joints [-0.003, -90.003, 0.004, -89.999, -0.001, 0] deg
              Call Quitar_Broca_Chida
              Call Poner_Broca
              MoveJ speed 60 deg/s, acceleration 80 deg/s^2 (useActiveTCP=true) feature=Base
                Waypoint Posicion_Cero: TCP in base x=0.551 y=-324.742 z=1651.532 mm, rx=-0.0041 ry=-0.0154 rz=-3.05 rad; joints [-0.003, -90.003, 0.004, -89.999, -0.001, 0] deg
                Waypoint Zona_izq1: TCP in base x=721.637 y=-174.262 z=505.425 mm, rx=2.3235 ry=2.1144 rz=0.0001 rad; joints [0.067, -89.734, -90.405, -179.332, -89.71, -0.034] deg
            ElseIf barrenoActual≟27
              MoveDirectionNode (selectedDirection=ZPlus)
                Until DISTANCE (allowActions=false deceleration=3 distanceNodeType=STOP) Distance=0.03; motionParameters(blendRadius=0)
              MoveJ speed 60 deg/s, acceleration 80 deg/s^2 (useActiveTCP=true) feature=Base
                Waypoint Zona_izq1: TCP in base x=721.637 y=-174.262 z=505.425 mm, rx=2.3235 ry=2.1144 rz=0.0001 rad; joints [0.067, -89.734, -90.405, -179.332, -89.71, -0.034] deg
                Waypoint Posicion_Cero: TCP in base x=0.551 y=-324.742 z=1651.532 mm, rx=-0.0041 ry=-0.0154 rz=-3.05 rad; joints [-0.003, -90.003, 0.004, -89.999, -0.001, 0] deg
              Call Quitar_Broca_Chida
              Set DigitalOutput pin=carrusel_home; digitalValue=1
              Wait Sleep waitTime=1
              Set DigitalOutput pin=carrusel_home; digitalValue=0
              Set ExpressionOutput pin=mensaje_mw10; expression=85
              Wait DigitalInput pin=Continuar_M30; digitalValue=1
              Wait Sleep waitTime=1
              Set ExpressionOutput pin=mensaje_mw10; expression=120
              Wait DigitalInput pin=Continuar_M30; digitalValue=1
              Wait Sleep waitTime=1
              Set DigitalOutput pin=carrusel_home; digitalValue=1
              Wait Sleep waitTime=1
              Set DigitalOutput pin=carrusel_home; digitalValue=0
              Set ExpressionOutput pin=mensaje_mw10; expression=90
              Wait DigitalInput pin=Continuar_M30; digitalValue=1
              Wait Sleep waitTime=1
              Call Poner_Broca
              broca := 217
              MoveJ speed 60 deg/s, acceleration 80 deg/s^2 (useActiveTCP=true) feature=Base
                Waypoint Posicion_Cero: TCP in base x=0.551 y=-324.742 z=1651.532 mm, rx=-0.0041 ry=-0.0154 rz=-3.05 rad; joints [-0.003, -90.003, 0.004, -89.999, -0.001, 0] deg
                Waypoint Zona_izq1: TCP in base x=721.637 y=-174.262 z=505.425 mm, rx=2.3235 ry=2.1144 rz=0.0001 rad; joints [0.067, -89.734, -90.405, -179.332, -89.71, -0.034] deg
              Set ExpressionOutput pin=mensaje_mw10; expression=95
              Wait DigitalInput pin=Continuar_M30; digitalValue=1
              Wait Sleep waitTime=1
              Set ExpressionOutput pin=mensaje_mw10; expression=150
              Wait DigitalInput pin=Continuar_M30; digitalValue=1
              Wait Sleep waitTime=1
            barrenoActual := barrenoActual+1
      Folder Linea 1 a 217
        broca := 217
        Folder Buje_inicial
          Buje_Inicial := L1B2
        Folder Buje_final
          Buje_Final := L1B1
        barrenosTotales := 27
        barrenoActual := 1
        Loop While (checkContinuously=false) expression=barrenoActual≤barrenosTotales
          MoveL speed 250 mm/s, acceleration 1200 mm/s^2 (useActiveTCP=true) feature=Base
            bajada_broca := p[0,0,0.018,0,0,0]
            internos := interpolate_pose(Buje_Inicial, Buje_Final, ((barrenoActual)-1)/((barrenosTotales)-1))
            Folder Alturas
              If barrenoActual≟3 or barrenoActual≟5 or barrenoActual≟7 or barrenoActual≟9 or barrenoActual≟11 or barrenoActual≟13 or barrenoActual≟15 or barrenoActual≟17 or barrenoActual≟19 or barrenoActual≟21 or barrenoActual≟23 or barrenoActual≟25 or barrenoActual≟27 or barrenoActual≟1
                Set ExpressionOutput pin=mensaje_mw10; expression=200
                Wait DigitalInput pin=Continuar_M30; digitalValue=1
                Wait Sleep waitTime=1
                Set ExpressionOutput pin=mensaje_mw10; expression=150
                Wait Sleep waitTime=1
              MoveJ speed 60 deg/s, acceleration 80 deg/s^2 (useActiveTCP=true) feature=Base
                Waypoint Waypoint (Variable): variable=internos
              Wait Sleep waitTime=2
              If P1h[2]<P2h[2]
                acomodin := (altura/(barrenosTotales-1))*(barrenoActual-1)
                tcp_chido := get_actual_tcp_pose()
                offset_bajada := p[tcp_chido[0],tcp_chido[1],((alta-0.0095)-(acomodin/1000)),tcp_chido[3],tcp_chido[4],tcp_chido[5]]
                MoveL speed 15 mm/s, acceleration 30 mm/s^2 (useActiveTCP=true) feature=Base
                  Waypoint Waypoint (Variable): variable=offset_bajada
              Else 
                acomodin := (altura/(barrenosTotales-1))*(26-(barrenoActual-1))
                tcp_chido := get_actual_tcp_pose()
                offset_bajada := p[tcp_chido[0],tcp_chido[1],((alta-0.0095)-(acomodin/1000)),tcp_chido[3],tcp_chido[4],tcp_chido[5]]
                MoveL speed 15 mm/s, acceleration 30 mm/s^2 (useActiveTCP=true) feature=Base
                  Waypoint Waypoint (Variable): variable=offset_bajada
            Folder Freemove
              Wait Sleep waitTime=2
              Script: freedrive_mode()
              Wait Sleep waitTime=2.5
              Script: end_freedrive_mode()
            Wait Sleep waitTime=0.3
            Set DigitalOutput pin=config_out[1]; digitalValue=1
            Wait Sleep waitTime=1
            Wait Sleep waitTime=0.3
            Wait Sleep waitTime=0.3
            Wait Sleep waitTime=0.3
            Loop Counting (count=1) loopVariable(name=Loop_19)
              Poses_taladrado := pose_sub(get_actual_tcp_pose(), bajada_broca)
              Waypoint Waypoint (Variable): motionParameters(jointSpeed=1.047198 jointAcceleration=1.396263 cartesianSpeed=0.001 cartesianAcceleration=0.005); variable=Poses_taladrado
              If bajada_broca≟p[0,0,0.018,0,0,0]
                num_barreno := str_cat("Barreno: ",barrenoActual)
                tcp_actual := get_actual_tcp_pose()
                X_actual := str_cat("     X: ",tcp_actual[0])
                Y_actual := str_cat("     Y: ",tcp_actual[1])
                pos_barreno := str_cat(X_actual,Y_actual)
                Script: textmsg(num_barreno,pos_barreno)
              Poses_taladrado := pose_add(get_actual_tcp_pose(), bajada_broca)
              Waypoint Waypoint (Variable): motionParameters(jointSpeed=1.047198 jointAcceleration=1.396263 cartesianSpeed=0.01 cartesianAcceleration=0.01); variable=Poses_taladrado
              bajada_broca := pose_add(bajada_broca, p[0,0,0.018,0,0,0])
            MoveDirectionNode (selectedDirection=ZPlus toolParams=0.03, 0.04)
              Until DISTANCE (allowActions=false deceleration=3 distanceNodeType=STOP) Distance=0.05; motionParameters(blendRadius=0)
            MoveJ speed 60 deg/s, acceleration 80 deg/s^2 (useActiveTCP=true) feature=Base
              Waypoint Waypoint (Variable): variable=internos
            Wait Sleep waitTime=0.3
            Set DigitalOutput pin=config_out[1]; digitalValue=0
            Wait Sleep waitTime=0.3
            If barrenoActual≟13 or barrenoActual≟27
              MoveDirectionNode (selectedDirection=ZPlus)
                Until DISTANCE (allowActions=false deceleration=3 distanceNodeType=STOP) Distance=0.03; motionParameters(blendRadius=0)
              MoveJ speed 60 deg/s, acceleration 80 deg/s^2 (useActiveTCP=true) feature=Base
                Waypoint Zona_izq1: TCP in base x=721.637 y=-174.262 z=505.425 mm, rx=2.3235 ry=2.1144 rz=0.0001 rad; joints [0.067, -89.734, -90.405, -179.332, -89.71, -0.034] deg
                Waypoint Posicion_Cero: TCP in base x=0.551 y=-324.742 z=1651.532 mm, rx=-0.0041 ry=-0.0154 rz=-3.05 rad; joints [-0.003, -90.003, 0.004, -89.999, -0.001, 0] deg
              Call Quitar_Broca_Chida
              Call Poner_Broca
              MoveJ speed 60 deg/s, acceleration 80 deg/s^2 (useActiveTCP=true) feature=Base
                Waypoint Posicion_Cero: TCP in base x=0.551 y=-324.742 z=1651.532 mm, rx=-0.0041 ry=-0.0154 rz=-3.05 rad; joints [-0.003, -90.003, 0.004, -89.999, -0.001, 0] deg
                Waypoint Zona_izq1: TCP in base x=721.637 y=-174.262 z=505.425 mm, rx=2.3235 ry=2.1144 rz=0.0001 rad; joints [0.067, -89.734, -90.405, -179.332, -89.71, -0.034] deg
            barrenoActual := barrenoActual+1
      Folder Linea 2 a 217
        broca := 217
        Folder Buje_inicial
          Buje_Inicial := L2B2
        Folder Buje_final
          Buje_Final := L2B1
        barrenosTotales := 27
        barrenoActual := 1
        Loop While (checkContinuously=false) expression=barrenoActual≤barrenosTotales
          MoveL speed 250 mm/s, acceleration 1200 mm/s^2 (useActiveTCP=true) feature=Base
            bajada_broca := p[0,0,0.018,0,0,0]
            internos := interpolate_pose(Buje_Inicial, Buje_Final, ((barrenoActual)-1)/((barrenosTotales)-1))
            Folder Alturas
              If barrenoActual≟3 or barrenoActual≟5 or barrenoActual≟7 or barrenoActual≟9 or barrenoActual≟11 or barrenoActual≟13 or barrenoActual≟15 or barrenoActual≟17 or barrenoActual≟19 or barrenoActual≟21 or barrenoActual≟23 or barrenoActual≟25 or barrenoActual≟27 or barrenoActual≟1
                Set ExpressionOutput pin=mensaje_mw10; expression=200
                Wait DigitalInput pin=Continuar_M30; digitalValue=1
                Wait Sleep waitTime=1
                Set ExpressionOutput pin=mensaje_mw10; expression=150
                Wait Sleep waitTime=1
              MoveJ speed 60 deg/s, acceleration 80 deg/s^2 (useActiveTCP=true) feature=Base
                Waypoint Waypoint (Variable): variable=internos
              Wait Sleep waitTime=2
              If P1h[2]<P2h[2]
                acomodin := (altura/(barrenosTotales-1))*(barrenoActual-1)
                tcp_chido := get_actual_tcp_pose()
                offset_bajada := p[tcp_chido[0],tcp_chido[1],((alta-0.0095)-(acomodin/1000)),tcp_chido[3],tcp_chido[4],tcp_chido[5]]
                MoveL speed 15 mm/s, acceleration 30 mm/s^2 (useActiveTCP=true) feature=Base
                  Waypoint Waypoint (Variable): variable=offset_bajada
              Else 
                acomodin := (altura/(barrenosTotales-1))*(26-(barrenoActual-1))
                tcp_chido := get_actual_tcp_pose()
                offset_bajada := p[tcp_chido[0],tcp_chido[1],((alta-0.0095)-(acomodin/1000)),tcp_chido[3],tcp_chido[4],tcp_chido[5]]
                MoveL speed 15 mm/s, acceleration 30 mm/s^2 (useActiveTCP=true) feature=Base
                  Waypoint Waypoint (Variable): variable=offset_bajada
            Folder Freemove
              Wait Sleep waitTime=2
              Script: freedrive_mode()
              Wait Sleep waitTime=2.5
              Script: end_freedrive_mode()
            Wait Sleep waitTime=0.3
            Set DigitalOutput pin=config_out[1]; digitalValue=1
            Wait Sleep waitTime=1
            Wait Sleep waitTime=0.3
            Wait Sleep waitTime=0.3
            Wait Sleep waitTime=0.3
            Loop Counting (count=1) loopVariable(name=Loop_21)
              Poses_taladrado := pose_sub(get_actual_tcp_pose(), bajada_broca)
              Waypoint Waypoint (Variable): motionParameters(jointSpeed=1.047198 jointAcceleration=1.396263 cartesianSpeed=0.001 cartesianAcceleration=0.005); variable=Poses_taladrado
              If bajada_broca≟p[0,0,0.018,0,0,0]
                num_barreno := str_cat("Barreno: ",barrenoActual)
                tcp_actual := get_actual_tcp_pose()
                X_actual := str_cat("     X: ",tcp_actual[0])
                Y_actual := str_cat("     Y: ",tcp_actual[1])
                pos_barreno := str_cat(X_actual,Y_actual)
                Script: textmsg(num_barreno,pos_barreno)
              Poses_taladrado := pose_add(get_actual_tcp_pose(), bajada_broca)
              Waypoint Waypoint (Variable): motionParameters(jointSpeed=1.047198 jointAcceleration=1.396263 cartesianSpeed=0.01 cartesianAcceleration=0.01); variable=Poses_taladrado
              bajada_broca := pose_add(bajada_broca, p[0,0,0.018,0,0,0])
            MoveDirectionNode (selectedDirection=ZPlus toolParams=0.03, 0.04)
              Until DISTANCE (allowActions=false deceleration=3 distanceNodeType=STOP) Distance=0.05; motionParameters(blendRadius=0)
            MoveJ speed 60 deg/s, acceleration 80 deg/s^2 (useActiveTCP=true) feature=Base
              Waypoint Waypoint (Variable): variable=internos
            Wait Sleep waitTime=0.3
            Set DigitalOutput pin=config_out[1]; digitalValue=0
            Wait Sleep waitTime=0.3
            If barrenoActual≟13
              MoveDirectionNode (selectedDirection=ZPlus)
                Until DISTANCE (allowActions=false deceleration=3 distanceNodeType=STOP) Distance=0.03; motionParameters(blendRadius=0)
              MoveJ speed 60 deg/s, acceleration 80 deg/s^2 (useActiveTCP=true) feature=Base
                Waypoint Zona_izq1: TCP in base x=721.637 y=-174.262 z=505.425 mm, rx=2.3235 ry=2.1144 rz=0.0001 rad; joints [0.067, -89.734, -90.405, -179.332, -89.71, -0.034] deg
                Waypoint Posicion_Cero: TCP in base x=0.551 y=-324.742 z=1651.532 mm, rx=-0.0041 ry=-0.0154 rz=-3.05 rad; joints [-0.003, -90.003, 0.004, -89.999, -0.001, 0] deg
              Call Quitar_Broca_Chida
              Call Poner_Broca
              MoveJ speed 60 deg/s, acceleration 80 deg/s^2 (useActiveTCP=true) feature=Base
                Waypoint Posicion_Cero: TCP in base x=0.551 y=-324.742 z=1651.532 mm, rx=-0.0041 ry=-0.0154 rz=-3.05 rad; joints [-0.003, -90.003, 0.004, -89.999, -0.001, 0] deg
                Waypoint Zona_izq1: TCP in base x=721.637 y=-174.262 z=505.425 mm, rx=2.3235 ry=2.1144 rz=0.0001 rad; joints [0.067, -89.734, -90.405, -179.332, -89.71, -0.034] deg
            ElseIf barrenoActual≟27
              MoveDirectionNode (selectedDirection=ZPlus)
                Until DISTANCE (allowActions=false deceleration=3 distanceNodeType=STOP) Distance=0.03; motionParameters(blendRadius=0)
              MoveJ speed 60 deg/s, acceleration 80 deg/s^2 (useActiveTCP=true) feature=Base
                Waypoint Zona_izq1: TCP in base x=721.637 y=-174.262 z=505.425 mm, rx=2.3235 ry=2.1144 rz=0.0001 rad; joints [0.067, -89.734, -90.405, -179.332, -89.71, -0.034] deg
                Waypoint Posicion_Cero: TCP in base x=0.551 y=-324.742 z=1651.532 mm, rx=-0.0041 ry=-0.0154 rz=-3.05 rad; joints [-0.003, -90.003, 0.004, -89.999, -0.001, 0] deg
              Call Quitar_Broca_Chida
              Set DigitalOutput pin=carrusel_home; digitalValue=1
              Wait Sleep waitTime=1
              Set DigitalOutput pin=carrusel_home; digitalValue=0
              Set ExpressionOutput pin=mensaje_mw10; expression=120
              Wait DigitalInput pin=Continuar_M30; digitalValue=1
              Wait Sleep waitTime=1
              Set ExpressionOutput pin=mensaje_mw10; expression=100
              Wait DigitalInput pin=Continuar_M30; digitalValue=1
              Wait Sleep waitTime=1
              MoveJ speed 60 deg/s, acceleration 80 deg/s^2 (useActiveTCP=true) feature=Base
                Waypoint Traslacion_izq: TCP in base x=-174.237 y=-721.63 z=505.386 mm, rx=-3.1292 ry=0.1412 rz=-0.0002 rad; joints [-90, -90.001, -90.002, -180, -90.003, -0.001] deg
            barrenoActual := barrenoActual+1
    SuppressedNode
      'Seatracks traseros listos'
    Folder Traslacion
      MoveJ speed 60 deg/s, acceleration 80 deg/s^2 (useActiveTCP=true) feature=Base
        Waypoint Traslacion_izq: TCP in base x=-174.237 y=-721.63 z=505.386 mm, rx=-3.1292 ry=0.1412 rz=-0.0002 rad; joints [-90, -90.001, -90.002, -180, -90.003, -0.001] deg
      Set ExpressionOutput pin=mensaje_mw10; expression=105
      Wait DigitalInput pin=Continuar_M30; digitalValue=1
      Wait Sleep waitTime=1
      Set ExpressionOutput pin=mensaje_mw10; expression=145
      Wait DigitalInput pin=Continuar_M30; digitalValue=1
      Wait Sleep waitTime=1
      Set DigitalOutput pin=postrnas_m187; digitalValue=1
      Wait Sleep waitTime=1
      Set DigitalOutput pin=pos2_izq_m697; digitalValue=1
      Wait Sleep waitTime=1
      Set DigitalOutput pin=pos2_izq_m697; digitalValue=0
      Set DigitalOutput pin=postrnas_m187; digitalValue=0
      Wait Sleep waitTime=5
    Folder Brocas
      Set DigitalOutput pin=carrusel_home; digitalValue=1
      Wait Sleep waitTime=1
      Set DigitalOutput pin=carrusel_home; digitalValue=0
      Set ExpressionOutput pin=mensaje_mw10; expression=40
      Wait DigitalInput pin=Continuar_M30; digitalValue=1
      Wait Sleep waitTime=1
      Set DigitalOutput pin=carrusel_home; digitalValue=1
      Wait Sleep waitTime=1
      Set DigitalOutput pin=carrusel_home; digitalValue=0
      Set ExpressionOutput pin=mensaje_mw10; expression=45
      Wait DigitalInput pin=Continuar_M30; digitalValue=1
      Wait Sleep waitTime=1
      Call Poner_Broca
    Folder Offsets factor
      SuppressedNode
        broca := 1645
      L1B1x := ((0.09523476)/(0.09525))*(0.09523476)
      L1B1y := ((-0.01278382)/(-0.0127))*(-0.01278382)
      L1B2x := ((0.75575414)/(0.75565))*(0.75575414)
      L1B2y := ((-0.01279398)/(-0.0127))*(-0.01279398)
      L2B1x := ((0.09675299)/(0.09525))*(0.09675299)
      L2B1y := ((0.3937)/(0.3937))*(0.3937)
      L2B2x := ((0.757306777)/(0.75565))*(0.757306777)
      L2B2y := ((0.393684081)/(0.3937))*(0.393684081)
    Folder Calibracion
      Set ExpressionOutput pin=mensaje_mw10; expression=50
      Wait DigitalInput pin=Continuar_M30; digitalValue=1
      Wait Sleep waitTime=1
      MoveJ speed 60 deg/s, acceleration 80 deg/s^2 (useActiveTCP=true) feature=Base
        Waypoint Posicion_Cero: TCP in base x=0.551 y=-324.742 z=1651.532 mm, rx=-0.0041 ry=-0.0154 rz=-3.05 rad; joints [-0.003, -90.003, 0.004, -89.999, -0.001, 0] deg
        Waypoint Zona_izq1: TCP in base x=721.637 y=-174.262 z=505.425 mm, rx=2.3235 ry=2.1144 rz=0.0001 rad; joints [0.067, -89.734, -90.405, -179.332, -89.71, -0.034] deg
      broca := 1645
      Set ExpressionOutput pin=mensaje_mw10; expression=125
      Wait DigitalInput pin=Continuar_M30; digitalValue=1
      Wait Sleep waitTime=1
      Set ExpressionOutput pin=mensaje_mw10; expression=130
      Wait DigitalInput pin=Continuar_M30; digitalValue=1
      Wait Sleep waitTime=1
      Call Calibracion
    Folder GoNoGo
      Set ExpressionOutput pin=mensaje_mw10; expression=55
      Wait DigitalInput pin=Continuar_M30; digitalValue=1
      Wait Sleep waitTime=1
      Set ExpressionOutput pin=mensaje_mw10; expression=60
      Wait DigitalInput pin=Continuar_M30; digitalValue=1
      Wait Sleep waitTime=1
      Folder Linea1_Buje1
        Xfin := ((((L1B1x)*(-1)*Xp)-(Xd)-((L1B1y)*(1/m2)))*(-1))*(1)
        Yfin := ((((L1B1y)*(-1)*Yp)-(Yd)+((L1B1x)*(-1)*m1))*(-1))*(1)
        rotaciones := get_actual_tcp_pose()
        var_3 := rotaciones[3]
        var_4 := rotaciones[4]
        var_5 := rotaciones[5]
        If broca≟1645
          PosFinal := p[Xfin-0.00208915,Yfin-0.00208915,0.15,var_3,var_4,var_5]
        ElseIf broca≟1935
          PosFinal := p[Xfin-0.00245745,Yfin-0.00245745,0.15,var_3,var_4,var_5]
        ElseIf broca≟217
          PosFinal := p[Xfin-0.0027559,Yfin-0.0027559,0.15,var_3,var_4,var_5]
        Buje_Final := PosFinal
      MoveJ speed 60 deg/s, acceleration 80 deg/s^2 (useActiveTCP=true) feature=Base
        Waypoint Waypoint (Variable): variable=Buje_Final
      Wait Sleep waitTime=1
      Folder Alturas
        If P1h[2]<P2h[2]
          tcp_chido := get_actual_tcp_pose()
          offset_bajada := p[tcp_chido[0],tcp_chido[1],((alta-0.0095)-(altura/1000)),tcp_chido[3],tcp_chido[4],tcp_chido[5]]
          MoveL speed 15 mm/s, acceleration 30 mm/s^2 (useActiveTCP=true) feature=Base
            Waypoint Waypoint (Variable): variable=offset_bajada
        Else 
          tcp_chido := get_actual_tcp_pose()
          offset_bajada := p[tcp_chido[0],tcp_chido[1],((alta-0.0095)),tcp_chido[3],tcp_chido[4],tcp_chido[5]]
          MoveL speed 15 mm/s, acceleration 30 mm/s^2 (useActiveTCP=true) feature=Base
            Waypoint Waypoint (Variable): variable=offset_bajada
      MoveL speed 15 mm/s, acceleration 30 mm/s^2 (useActiveTCP=true) feature=Base
        Folder Freemove
          Wait Sleep waitTime=2
          Script: freedrive_mode()
          Wait Sleep waitTime=2.5
          Script: end_freedrive_mode()
          var_13 := get_actual_tcp_pose()
          var_13 := p[var_13[0]*1000,var_13[1]*1000,420,420,420,420]
          var_13 := get_actual_tcp_pose()
          var_13 := p[var_13[0],var_13[1],0.1,var_13[3],var_13[4],var_13[5]]
        MoveDirectionNode (selectedDirection=ZPlus)
          Until DISTANCE (allowActions=false deceleration=3 distanceNodeType=STOP) Distance=0.15; motionParameters(blendRadius=0)
      L1B1 := var_13
      Folder Linea1_Buje2
        Xfin := ((((L1B2x)*(-1)*Xp)-(Xd)-((L1B2y)*(1/m2)))*(-1))*(1)
        Yfin := ((((L1B2y)*(-1)*Yp)-(Yd)+((L1B2x)*(-1)*m1))*(-1))*(1)
        rotaciones := get_actual_tcp_pose()
        var_3 := rotaciones[3]
        var_4 := rotaciones[4]
        var_5 := rotaciones[5]
        If broca≟1645
          PosFinal := p[Xfin-0.00208915,Yfin-0.00208915,0.15,var_3,var_4,var_5]
        ElseIf broca≟1935
          PosFinal := p[Xfin-0.00245745,Yfin-0.00245745,0.15,var_3,var_4,var_5]
        ElseIf broca≟217
          PosFinal := p[Xfin-0.0027559,Yfin-0.0027559,0.15,var_3,var_4,var_5]
        Buje_Final := PosFinal
      MoveJ speed 60 deg/s, acceleration 80 deg/s^2 (useActiveTCP=true) feature=Base
        Waypoint Waypoint (Variable): variable=Buje_Final
      Wait Sleep waitTime=1
      Folder Alturas
        If P1h[2]<P2h[2]
          tcp_chido := get_actual_tcp_pose()
          offset_bajada := p[tcp_chido[0],tcp_chido[1],((alta-0.0095)),tcp_chido[3],tcp_chido[4],tcp_chido[5]]
          MoveL speed 15 mm/s, acceleration 30 mm/s^2 (useActiveTCP=true) feature=Base
            Waypoint Waypoint (Variable): variable=offset_bajada
        Else 
          tcp_chido := get_actual_tcp_pose()
          offset_bajada := p[tcp_chido[0],tcp_chido[1],((alta-0.0095)-(altura/1000)),tcp_chido[3],tcp_chido[4],tcp_chido[5]]
          MoveL speed 15 mm/s, acceleration 30 mm/s^2 (useActiveTCP=true) feature=Base
            Waypoint Waypoint (Variable): variable=offset_bajada
      MoveL speed 15 mm/s, acceleration 30 mm/s^2 (useActiveTCP=true) feature=Base
        Folder Freemove
          Wait Sleep waitTime=2
          Script: freedrive_mode()
          Wait Sleep waitTime=2.5
          Script: end_freedrive_mode()
          var_13 := get_actual_tcp_pose()
          var_13 := p[var_13[0]*1000,var_13[1]*1000,420,420,420,420]
          var_13 := get_actual_tcp_pose()
          var_13 := p[var_13[0],var_13[1],0.1,var_13[3],var_13[4],var_13[5]]
        MoveDirectionNode (selectedDirection=ZPlus)
          Until DISTANCE (allowActions=false deceleration=3 distanceNodeType=STOP) Distance=0.15; motionParameters(blendRadius=0)
      L1B2 := var_13
      Folder Linea2_Buje2
        Xfin := ((((L2B2x)*(-1)*Xp)-(Xd)-(L2B2y*(1/m2)))*(-1))*(1)
        Yfin := ((((L2B2y)*(-1)*Yp)-(Yd)+((L2B2x)*(-1)*m1))*(-1))*(1)
        rotaciones := get_actual_tcp_pose()
        var_3 := rotaciones[3]
        var_4 := rotaciones[4]
        var_5 := rotaciones[5]
        If broca≟1645
          PosFinal := p[Xfin-0.00208915,Yfin-0.00208915,0.15,var_3,var_4,var_5]
        ElseIf broca≟1935
          PosFinal := p[Xfin-0.00245745,Yfin-0.00245745,0.15,var_3,var_4,var_5]
        ElseIf broca≟217
          PosFinal := p[Xfin-0.0027559,Yfin-0.0027559,0.15,var_3,var_4,var_5]
        Buje_Final := PosFinal
      MoveJ speed 60 deg/s, acceleration 80 deg/s^2 (useActiveTCP=true) feature=Base
        Waypoint Waypoint (Variable): variable=Buje_Final
      Wait Sleep waitTime=1
      Folder Alturas
        If P1h[2]<P2h[2]
          tcp_chido := get_actual_tcp_pose()
          offset_bajada := p[tcp_chido[0],tcp_chido[1],((alta-0.0095)),tcp_chido[3],tcp_chido[4],tcp_chido[5]]
          MoveL speed 15 mm/s, acceleration 30 mm/s^2 (useActiveTCP=true) feature=Base
            Waypoint Waypoint (Variable): variable=offset_bajada
        Else 
          tcp_chido := get_actual_tcp_pose()
          offset_bajada := p[tcp_chido[0],tcp_chido[1],((alta-0.0095)-(altura/1000)),tcp_chido[3],tcp_chido[4],tcp_chido[5]]
          MoveL speed 15 mm/s, acceleration 30 mm/s^2 (useActiveTCP=true) feature=Base
            Waypoint Waypoint (Variable): variable=offset_bajada
      MoveL speed 15 mm/s, acceleration 30 mm/s^2 (useActiveTCP=true) feature=Base
        Folder Freemove
          Wait Sleep waitTime=2
          Script: freedrive_mode()
          Wait Sleep waitTime=2.5
          Script: end_freedrive_mode()
          var_13 := get_actual_tcp_pose()
          var_13 := p[var_13[0]*1000,var_13[1]*1000,420,420,420,420]
          var_13 := get_actual_tcp_pose()
          var_13 := p[var_13[0],var_13[1],0.1,var_13[3],var_13[4],var_13[5]]
        MoveDirectionNode (selectedDirection=ZPlus)
          Until DISTANCE (allowActions=false deceleration=3 distanceNodeType=STOP) Distance=0.15; motionParameters(blendRadius=0)
      L2B2 := var_13
      Folder Linea2_Buje1
        Xfin := ((((L2B1x)*(-1)*Xp)-(Xd)-((L2B1y)*(1/m2)))*(-1))*(1)
        Yfin := ((((L2B1y)*(-1)*Yp)-(Yd)+((L2B1x)*(-1)*m1))*(-1))*(1)
        rotaciones := get_actual_tcp_pose()
        var_3 := rotaciones[3]
        var_4 := rotaciones[4]
        var_5 := rotaciones[5]
        If broca≟1645
          PosFinal := p[Xfin-0.00208915,Yfin-0.00208915,0.15,var_3,var_4,var_5]
        ElseIf broca≟1935
          PosFinal := p[Xfin-0.00245745,Yfin-0.00245745,0.15,var_3,var_4,var_5]
        ElseIf broca≟217
          PosFinal := p[Xfin-0.0027559,Yfin-0.0027559,0.15,var_3,var_4,var_5]
        Buje_Final := PosFinal
      MoveJ speed 60 deg/s, acceleration 80 deg/s^2 (useActiveTCP=true) feature=Base
        Waypoint Paso2_izq1: TCP in base x=414.118 y=-280.673 z=89.978 mm, rx=-2.3928 ry=-2.0356 rz=0 rad; joints [-18.236, -84.335, -142.099, -133.065, -104.295, 0.11] deg
        Waypoint Waypoint (Variable): variable=Buje_Final
      Wait Sleep waitTime=1
      Folder Alturas
        If P1h[2]<P2h[2]
          tcp_chido := get_actual_tcp_pose()
          offset_bajada := p[tcp_chido[0],tcp_chido[1],((alta-0.0095)-(altura/1000)),tcp_chido[3],tcp_chido[4],tcp_chido[5]]
          MoveL speed 15 mm/s, acceleration 30 mm/s^2 (useActiveTCP=true) feature=Base
            Waypoint Waypoint (Variable): variable=offset_bajada
        Else 
          tcp_chido := get_actual_tcp_pose()
          offset_bajada := p[tcp_chido[0],tcp_chido[1],((alta-0.0095)),tcp_chido[3],tcp_chido[4],tcp_chido[5]]
          MoveL speed 15 mm/s, acceleration 30 mm/s^2 (useActiveTCP=true) feature=Base
            Waypoint Waypoint (Variable): variable=offset_bajada
      MoveL speed 15 mm/s, acceleration 30 mm/s^2 (useActiveTCP=true) feature=Base
        Folder Freemove
          Wait Sleep waitTime=2
          Script: freedrive_mode()
          Wait Sleep waitTime=2.5
          Script: end_freedrive_mode()
          var_13 := get_actual_tcp_pose()
          var_13 := p[var_13[0]*1000,var_13[1]*1000,420,420,420,420]
          var_13 := get_actual_tcp_pose()
          var_13 := p[var_13[0],var_13[1],0.1,var_13[3],var_13[4],var_13[5]]
        MoveDirectionNode (selectedDirection=ZPlus)
          Until DISTANCE (allowActions=false deceleration=3 distanceNodeType=STOP) Distance=0.15; motionParameters(blendRadius=0)
      MoveJ speed 60 deg/s, acceleration 80 deg/s^2 (useActiveTCP=true) feature=Base
        Waypoint Zona_izq1: TCP in base x=721.637 y=-174.262 z=505.425 mm, rx=2.3235 ry=2.1144 rz=0.0001 rad; joints [0.067, -89.734, -90.405, -179.332, -89.71, -0.034] deg
      L2B1 := var_13
    SuppressedNode
      Folder Cancelar barrenado
        MoveJ speed 60 deg/s, acceleration 80 deg/s^2 (useActiveTCP=true) feature=Base
          SuppressedNode
            Waypoint Zona_der1: TCP in base x=-724.618 y=-175.006 z=455.096 mm, rx=2.0346 ry=-2.3862 rz=-0.0105 rad; joints [0.001, -89.997, 90, 0.002, 90.001, 0.002] deg; TCP offset x=0.411 y=-218.298 z=37.994 mm, rx=1.558 ry=-0.1255 rz=0.1212 rad
          Waypoint Zona_izq1: TCP in base x=721.637 y=-174.262 z=505.425 mm, rx=2.3235 ry=2.1144 rz=0.0001 rad; joints [0.067, -89.734, -90.405, -179.332, -89.71, -0.034] deg; TCP offset x=0.151 y=-167.165 z=35.088 mm, rx=1.5784 ry=-0.0729 rz=0.0687 rad
          Waypoint Posicion_Cero: TCP in base x=0.551 y=-324.742 z=1651.532 mm, rx=-0.0041 ry=-0.0154 rz=-3.05 rad; joints [-0.003, -90.003, 0.004, -89.999, -0.001, 0] deg
        Call Quitar_Broca_Chida
        Set ExpressionOutput pin=mensaje_mw10; expression=100
        Wait DigitalInput pin=Continuar_M30; digitalValue=1
        Wait Sleep waitTime=1
        Set ExpressionOutput pin=mensaje_mw10; expression=155
        Wait DigitalInput pin=Continuar_M30; digitalValue=1
        Wait Sleep waitTime=1
    Folder Colocar broca
      Call Quitar_Broca_Chida
      Call Poner_Broca
    Folder Barrenado1
      Set ExpressionOutput pin=mensaje_mw10; expression=65
      Wait DigitalInput pin=Continuar_M30; digitalValue=1
      Wait Sleep waitTime=1
      Set ExpressionOutput pin=mensaje_mw10; expression=150
      Wait Sleep waitTime=1
      Folder Linea 1 a 1645
        broca := 1645
        Folder Buje_inicial
          Buje_Inicial := L1B2
        Folder Buje_final
          Buje_Final := L1B1
        barrenosTotales := 27
        barrenoActual := 1
        Loop While (checkContinuously=false) expression=barrenoActual≤barrenosTotales
          MoveL speed 250 mm/s, acceleration 1200 mm/s^2 (useActiveTCP=true) feature=Base
            bajada_broca := p[0,0,0.006,0,0,0]
            internos := interpolate_pose(Buje_Inicial, Buje_Final, ((barrenoActual)-1)/((barrenosTotales)-1))
            Folder Alturas
              If barrenoActual≟3 or barrenoActual≟5 or barrenoActual≟7 or barrenoActual≟9 or barrenoActual≟11 or barrenoActual≟13 or barrenoActual≟15 or barrenoActual≟17 or barrenoActual≟19 or barrenoActual≟21 or barrenoActual≟23 or barrenoActual≟25 or barrenoActual≟27 or barrenoActual≟1
                Set ExpressionOutput pin=mensaje_mw10; expression=200
                Wait DigitalInput pin=Continuar_M30; digitalValue=1
                Wait Sleep waitTime=1
                Set ExpressionOutput pin=mensaje_mw10; expression=150
                Wait Sleep waitTime=1
              MoveJ speed 60 deg/s, acceleration 80 deg/s^2 (useActiveTCP=true) feature=Base
                Waypoint Waypoint (Variable): variable=internos
              Wait Sleep waitTime=2
              If P1h[2]<P2h[2]
                acomodin := (altura/(barrenosTotales-1))*(barrenoActual-1)
                tcp_chido := get_actual_tcp_pose()
                offset_bajada := p[tcp_chido[0],tcp_chido[1],((alta-0.0095)-(acomodin/1000)),tcp_chido[3],tcp_chido[4],tcp_chido[5]]
                MoveL speed 15 mm/s, acceleration 30 mm/s^2 (useActiveTCP=true) feature=Base
                  Waypoint Waypoint (Variable): variable=offset_bajada
              Else 
                acomodin := (altura/(barrenosTotales-1))*(26-(barrenoActual-1))
                tcp_chido := get_actual_tcp_pose()
                offset_bajada := p[tcp_chido[0],tcp_chido[1],((alta-0.0095)-(acomodin/1000)),tcp_chido[3],tcp_chido[4],tcp_chido[5]]
                MoveL speed 15 mm/s, acceleration 30 mm/s^2 (useActiveTCP=true) feature=Base
                  Waypoint Waypoint (Variable): variable=offset_bajada
            Folder Freemove
              Wait Sleep waitTime=2
              Script: freedrive_mode()
              Wait Sleep waitTime=2.5
              Script: end_freedrive_mode()
            Wait Sleep waitTime=0.3
            Set DigitalOutput pin=config_out[1]; digitalValue=1
            Wait Sleep waitTime=1
            Wait Sleep waitTime=0.3
            Wait Sleep waitTime=0.3
            Wait Sleep waitTime=0.3
            Loop Counting (count=3) loopVariable(name=Loop_68)
              Poses_taladrado := pose_sub(get_actual_tcp_pose(), bajada_broca)
              Waypoint Waypoint (Variable): motionParameters(jointSpeed=1.047198 jointAcceleration=1.396263 cartesianSpeed=0.001 cartesianAcceleration=0.005); variable=Poses_taladrado
              If bajada_broca≟p[0,0,0.018,0,0,0]
                num_barreno := str_cat("Barreno: ",barrenoActual)
                tcp_actual := get_actual_tcp_pose()
                X_actual := str_cat("     X: ",tcp_actual[0])
                Y_actual := str_cat("     Y: ",tcp_actual[1])
                pos_barreno := str_cat(X_actual,Y_actual)
                Script: textmsg(num_barreno,pos_barreno)
              Poses_taladrado := pose_add(get_actual_tcp_pose(), bajada_broca)
              Waypoint Waypoint (Variable): motionParameters(jointSpeed=1.047198 jointAcceleration=1.396263 cartesianSpeed=0.01 cartesianAcceleration=0.01); variable=Poses_taladrado
              bajada_broca := pose_add(bajada_broca, p[0,0,0.006,0,0,0])
            MoveDirectionNode (selectedDirection=ZPlus toolParams=0.03, 0.04)
              Until DISTANCE (allowActions=false deceleration=3 distanceNodeType=STOP) Distance=0.05; motionParameters(blendRadius=0)
            MoveJ speed 60 deg/s, acceleration 80 deg/s^2 (useActiveTCP=true) feature=Base
              Waypoint Waypoint (Variable): variable=internos
            Wait Sleep waitTime=0.3
            Set DigitalOutput pin=config_out[1]; digitalValue=0
            Wait Sleep waitTime=0.3
            If barrenoActual≟13 or barrenoActual≟27
              MoveDirectionNode (selectedDirection=ZPlus toolParams=0.03, 0.04)
                Until DISTANCE (allowActions=false deceleration=3 distanceNodeType=STOP) Distance=0.03; motionParameters(blendRadius=0)
              MoveJ speed 60 deg/s, acceleration 80 deg/s^2 (useActiveTCP=true) feature=Base
                Waypoint Zona_izq1: TCP in base x=721.637 y=-174.262 z=505.425 mm, rx=2.3235 ry=2.1144 rz=0.0001 rad; joints [0.067, -89.734, -90.405, -179.332, -89.71, -0.034] deg
                Waypoint Posicion_Cero: TCP in base x=0.551 y=-324.742 z=1651.532 mm, rx=-0.0041 ry=-0.0154 rz=-3.05 rad; joints [-0.003, -90.003, 0.004, -89.999, -0.001, 0] deg
              Call Quitar_Broca_Chida
              Call Poner_Broca
              MoveJ speed 60 deg/s, acceleration 80 deg/s^2 (useActiveTCP=true) feature=Base
                Waypoint Posicion_Cero: TCP in base x=0.551 y=-324.742 z=1651.532 mm, rx=-0.0041 ry=-0.0154 rz=-3.05 rad; joints [-0.003, -90.003, 0.004, -89.999, -0.001, 0] deg
                Waypoint Zona_izq1: TCP in base x=721.637 y=-174.262 z=505.425 mm, rx=2.3235 ry=2.1144 rz=0.0001 rad; joints [0.067, -89.734, -90.405, -179.332, -89.71, -0.034] deg
            barrenoActual := barrenoActual+1
      Folder Linea 2 a 1645
        broca := 1645
        Folder Buje_inicial
          Buje_Inicial := L2B2
        Folder Buje_final
          Buje_Final := L2B1
        barrenosTotales := 27
        barrenoActual := 1
        Loop While (checkContinuously=false) expression=barrenoActual≤barrenosTotales
          MoveL speed 250 mm/s, acceleration 1200 mm/s^2 (useActiveTCP=true) feature=Base
            bajada_broca := p[0,0,0.006,0,0,0]
            internos := interpolate_pose(Buje_Inicial, Buje_Final, ((barrenoActual)-1)/((barrenosTotales)-1))
            Folder Alturas
              If barrenoActual≟3 or barrenoActual≟5 or barrenoActual≟7 or barrenoActual≟9 or barrenoActual≟11 or barrenoActual≟13 or barrenoActual≟15 or barrenoActual≟17 or barrenoActual≟19 or barrenoActual≟21 or barrenoActual≟23 or barrenoActual≟25 or barrenoActual≟27 or barrenoActual≟1
                Set ExpressionOutput pin=mensaje_mw10; expression=200
                Wait DigitalInput pin=Continuar_M30; digitalValue=1
                Wait Sleep waitTime=1
                Set ExpressionOutput pin=mensaje_mw10; expression=150
                Wait Sleep waitTime=1
              MoveJ speed 60 deg/s, acceleration 80 deg/s^2 (useActiveTCP=true) feature=Base
                Waypoint Waypoint (Variable): variable=internos
              Wait Sleep waitTime=2
              If P1h[2]<P2h[2]
                acomodin := (altura/(barrenosTotales-1))*(barrenoActual-1)
                tcp_chido := get_actual_tcp_pose()
                offset_bajada := p[tcp_chido[0],tcp_chido[1],((alta-0.0095)-(acomodin/1000)),tcp_chido[3],tcp_chido[4],tcp_chido[5]]
                MoveL speed 15 mm/s, acceleration 30 mm/s^2 (useActiveTCP=true) feature=Base
                  Waypoint Waypoint (Variable): variable=offset_bajada
              Else 
                acomodin := (altura/(barrenosTotales-1))*(26-(barrenoActual-1))
                tcp_chido := get_actual_tcp_pose()
                offset_bajada := p[tcp_chido[0],tcp_chido[1],((alta-0.0095)-(acomodin/1000)),tcp_chido[3],tcp_chido[4],tcp_chido[5]]
                MoveL speed 15 mm/s, acceleration 30 mm/s^2 (useActiveTCP=true) feature=Base
                  Waypoint Waypoint (Variable): variable=offset_bajada
            Folder Freemove
              Wait Sleep waitTime=2
              Script: freedrive_mode()
              Wait Sleep waitTime=2.5
              Script: end_freedrive_mode()
            Wait Sleep waitTime=0.3
            Set DigitalOutput pin=config_out[1]; digitalValue=1
            Wait Sleep waitTime=1
            Wait Sleep waitTime=0.3
            Wait Sleep waitTime=0.3
            Wait Sleep waitTime=0.3
            Loop Counting (count=3) loopVariable(name=Loop_70)
              Poses_taladrado := pose_sub(get_actual_tcp_pose(), bajada_broca)
              Waypoint Waypoint (Variable): motionParameters(jointSpeed=1.047198 jointAcceleration=1.396263 cartesianSpeed=0.001 cartesianAcceleration=0.005); variable=Poses_taladrado
              If bajada_broca≟p[0,0,0.018,0,0,0]
                num_barreno := str_cat("Barreno: ",barrenoActual)
                tcp_actual := get_actual_tcp_pose()
                X_actual := str_cat("     X: ",tcp_actual[0])
                Y_actual := str_cat("     Y: ",tcp_actual[1])
                pos_barreno := str_cat(X_actual,Y_actual)
                Script: textmsg(num_barreno,pos_barreno)
              Poses_taladrado := pose_add(get_actual_tcp_pose(), bajada_broca)
              Waypoint Waypoint (Variable): motionParameters(jointSpeed=1.047198 jointAcceleration=1.396263 cartesianSpeed=0.01 cartesianAcceleration=0.01); variable=Poses_taladrado
              bajada_broca := pose_add(bajada_broca, p[0,0,0.006,0,0,0])
            MoveDirectionNode (selectedDirection=ZPlus toolParams=0.03, 0.04)
              Until DISTANCE (allowActions=false deceleration=3 distanceNodeType=STOP) Distance=0.05; motionParameters(blendRadius=0)
            MoveJ speed 60 deg/s, acceleration 80 deg/s^2 (useActiveTCP=true) feature=Base
              Waypoint Waypoint (Variable): variable=internos
            Wait Sleep waitTime=0.3
            Set DigitalOutput pin=config_out[1]; digitalValue=0
            Wait Sleep waitTime=0.3
            If barrenoActual≟13
              MoveDirectionNode (selectedDirection=ZPlus)
                Until DISTANCE (allowActions=false deceleration=3 distanceNodeType=STOP) Distance=0.03; motionParameters(blendRadius=0)
              MoveJ speed 60 deg/s, acceleration 80 deg/s^2 (useActiveTCP=true) feature=Base
                Waypoint Zona_izq1: TCP in base x=721.637 y=-174.262 z=505.425 mm, rx=2.3235 ry=2.1144 rz=0.0001 rad; joints [0.067, -89.734, -90.405, -179.332, -89.71, -0.034] deg
                Waypoint Posicion_Cero: TCP in base x=0.551 y=-324.742 z=1651.532 mm, rx=-0.0041 ry=-0.0154 rz=-3.05 rad; joints [-0.003, -90.003, 0.004, -89.999, -0.001, 0] deg
              Call Quitar_Broca_Chida
              Call Poner_Broca
              MoveJ speed 60 deg/s, acceleration 80 deg/s^2 (useActiveTCP=true) feature=Base
                Waypoint Posicion_Cero: TCP in base x=0.551 y=-324.742 z=1651.532 mm, rx=-0.0041 ry=-0.0154 rz=-3.05 rad; joints [-0.003, -90.003, 0.004, -89.999, -0.001, 0] deg
                Waypoint Zona_izq1: TCP in base x=721.637 y=-174.262 z=505.425 mm, rx=2.3235 ry=2.1144 rz=0.0001 rad; joints [0.067, -89.734, -90.405, -179.332, -89.71, -0.034] deg
            ElseIf barrenoActual≟27
              MoveDirectionNode (selectedDirection=ZPlus)
                Until DISTANCE (allowActions=false deceleration=3 distanceNodeType=STOP) Distance=0.03; motionParameters(blendRadius=0)
              MoveJ speed 60 deg/s, acceleration 80 deg/s^2 (useActiveTCP=true) feature=Base
                Waypoint Zona_izq1: TCP in base x=721.637 y=-174.262 z=505.425 mm, rx=2.3235 ry=2.1144 rz=0.0001 rad; joints [0.067, -89.734, -90.405, -179.332, -89.71, -0.034] deg
                Waypoint Posicion_Cero: TCP in base x=0.551 y=-324.742 z=1651.532 mm, rx=-0.0041 ry=-0.0154 rz=-3.05 rad; joints [-0.003, -90.003, 0.004, -89.999, -0.001, 0] deg
              Call Quitar_Broca_Chida
              Set DigitalOutput pin=carrusel_home; digitalValue=1
              Wait Sleep waitTime=1
              Set DigitalOutput pin=carrusel_home; digitalValue=0
              Set ExpressionOutput pin=mensaje_mw10; expression=70
              Wait DigitalInput pin=Continuar_M30; digitalValue=1
              Wait Sleep waitTime=1
              Set ExpressionOutput pin=mensaje_mw10; expression=120
              Wait DigitalInput pin=Continuar_M30; digitalValue=1
              Wait Sleep waitTime=1
              Set DigitalOutput pin=carrusel_home; digitalValue=1
              Wait Sleep waitTime=1
              Set DigitalOutput pin=carrusel_home; digitalValue=0
              Set ExpressionOutput pin=mensaje_mw10; expression=75
              Wait DigitalInput pin=Continuar_M30; digitalValue=1
              Wait Sleep waitTime=1
              Call Poner_Broca
              broca := 1935
              MoveJ speed 60 deg/s, acceleration 80 deg/s^2 (useActiveTCP=true) feature=Base
                Waypoint Posicion_Cero: TCP in base x=0.551 y=-324.742 z=1651.532 mm, rx=-0.0041 ry=-0.0154 rz=-3.05 rad; joints [-0.003, -90.003, 0.004, -89.999, -0.001, 0] deg
                Waypoint Zona_izq1: TCP in base x=721.637 y=-174.262 z=505.425 mm, rx=2.3235 ry=2.1144 rz=0.0001 rad; joints [0.067, -89.734, -90.405, -179.332, -89.71, -0.034] deg
              Set ExpressionOutput pin=mensaje_mw10; expression=80
              Wait DigitalInput pin=Continuar_M30; digitalValue=1
              Wait Sleep waitTime=1
              Set ExpressionOutput pin=mensaje_mw10; expression=150
              Wait DigitalInput pin=Continuar_M30; digitalValue=1
              Wait Sleep waitTime=1
            barrenoActual := barrenoActual+1
      Folder Linea 1 a 1935
        broca := 1935
        Folder Buje_inicial
          Buje_Inicial := L1B2
        Folder Buje_final
          Buje_Final := L1B1
        barrenosTotales := 27
        barrenoActual := 1
        Loop While (checkContinuously=false) expression=barrenoActual≤barrenosTotales
          MoveL speed 250 mm/s, acceleration 1200 mm/s^2 (useActiveTCP=true) feature=Base
            bajada_broca := p[0,0,0.009,0,0,0]
            internos := interpolate_pose(Buje_Inicial, Buje_Final, ((barrenoActual)-1)/((barrenosTotales)-1))
            Folder Alturas
              If barrenoActual≟3 or barrenoActual≟5 or barrenoActual≟7 or barrenoActual≟9 or barrenoActual≟11 or barrenoActual≟13 or barrenoActual≟15 or barrenoActual≟17 or barrenoActual≟19 or barrenoActual≟21 or barrenoActual≟23 or barrenoActual≟25 or barrenoActual≟27 or barrenoActual≟1
                Set ExpressionOutput pin=mensaje_mw10; expression=200
                Wait DigitalInput pin=Continuar_M30; digitalValue=1
                Wait Sleep waitTime=1
                Set ExpressionOutput pin=mensaje_mw10; expression=150
                Wait Sleep waitTime=1
              MoveJ speed 60 deg/s, acceleration 80 deg/s^2 (useActiveTCP=true) feature=Base
                Waypoint Waypoint (Variable): variable=internos
              Wait Sleep waitTime=2
              If P1h[2]<P2h[2]
                acomodin := (altura/(barrenosTotales-1))*(barrenoActual-1)
                tcp_chido := get_actual_tcp_pose()
                offset_bajada := p[tcp_chido[0],tcp_chido[1],((alta-0.0095)-(acomodin/1000)),tcp_chido[3],tcp_chido[4],tcp_chido[5]]
                MoveL speed 15 mm/s, acceleration 30 mm/s^2 (useActiveTCP=true) feature=Base
                  Waypoint Waypoint (Variable): variable=offset_bajada
              Else 
                acomodin := (altura/(barrenosTotales-1))*(26-(barrenoActual-1))
                tcp_chido := get_actual_tcp_pose()
                offset_bajada := p[tcp_chido[0],tcp_chido[1],((alta-0.0095)-(acomodin/1000)),tcp_chido[3],tcp_chido[4],tcp_chido[5]]
                MoveL speed 15 mm/s, acceleration 30 mm/s^2 (useActiveTCP=true) feature=Base
                  Waypoint Waypoint (Variable): variable=offset_bajada
            Folder Freemove
              Wait Sleep waitTime=2
              Script: freedrive_mode()
              Wait Sleep waitTime=2.5
              Script: end_freedrive_mode()
            Wait Sleep waitTime=0.3
            Set DigitalOutput pin=config_out[1]; digitalValue=1
            Wait Sleep waitTime=1
            Wait Sleep waitTime=0.3
            Wait Sleep waitTime=0.3
            Wait Sleep waitTime=0.3
            Loop Counting (count=2) loopVariable(name=Loop_72)
              Poses_taladrado := pose_sub(get_actual_tcp_pose(), bajada_broca)
              Waypoint Waypoint (Variable): motionParameters(jointSpeed=1.047198 jointAcceleration=1.396263 cartesianSpeed=0.001 cartesianAcceleration=0.005); variable=Poses_taladrado
              If bajada_broca≟p[0,0,0.018,0,0,0]
                num_barreno := str_cat("Barreno: ",barrenoActual)
                tcp_actual := get_actual_tcp_pose()
                X_actual := str_cat("     X: ",tcp_actual[0])
                Y_actual := str_cat("     Y: ",tcp_actual[1])
                pos_barreno := str_cat(X_actual,Y_actual)
                Script: textmsg(num_barreno,pos_barreno)
              Poses_taladrado := pose_add(get_actual_tcp_pose(), bajada_broca)
              Waypoint Waypoint (Variable): motionParameters(jointSpeed=1.047198 jointAcceleration=1.396263 cartesianSpeed=0.01 cartesianAcceleration=0.01); variable=Poses_taladrado
              bajada_broca := pose_add(bajada_broca, p[0,0,0.009,0,0,0])
            MoveDirectionNode (selectedDirection=ZPlus toolParams=0.03, 0.04)
              Until DISTANCE (allowActions=false deceleration=3 distanceNodeType=STOP) Distance=0.05; motionParameters(blendRadius=0)
            MoveJ speed 60 deg/s, acceleration 80 deg/s^2 (useActiveTCP=true) feature=Base
              Waypoint Waypoint (Variable): variable=internos
            Wait Sleep waitTime=0.3
            Set DigitalOutput pin=config_out[1]; digitalValue=0
            Wait Sleep waitTime=0.3
            If barrenoActual≟13 or barrenoActual≟27
              MoveDirectionNode (selectedDirection=ZPlus)
                Until DISTANCE (allowActions=false deceleration=3 distanceNodeType=STOP) Distance=0.03; motionParameters(blendRadius=0)
              MoveJ speed 60 deg/s, acceleration 80 deg/s^2 (useActiveTCP=true) feature=Base
                Waypoint Zona_izq1: TCP in base x=721.637 y=-174.262 z=505.425 mm, rx=2.3235 ry=2.1144 rz=0.0001 rad; joints [0.067, -89.734, -90.405, -179.332, -89.71, -0.034] deg
                Waypoint Posicion_Cero: TCP in base x=0.551 y=-324.742 z=1651.532 mm, rx=-0.0041 ry=-0.0154 rz=-3.05 rad; joints [-0.003, -90.003, 0.004, -89.999, -0.001, 0] deg
              Call Quitar_Broca_Chida
              Call Poner_Broca
              MoveJ speed 60 deg/s, acceleration 80 deg/s^2 (useActiveTCP=true) feature=Base
                Waypoint Posicion_Cero: TCP in base x=0.551 y=-324.742 z=1651.532 mm, rx=-0.0041 ry=-0.0154 rz=-3.05 rad; joints [-0.003, -90.003, 0.004, -89.999, -0.001, 0] deg
                Waypoint Zona_izq1: TCP in base x=721.637 y=-174.262 z=505.425 mm, rx=2.3235 ry=2.1144 rz=0.0001 rad; joints [0.067, -89.734, -90.405, -179.332, -89.71, -0.034] deg
            barrenoActual := barrenoActual+1
      Folder Linea 2 a 1935
        broca := 1935
        Folder Buje_inicial
          Buje_Inicial := L2B2
        Folder Buje_final
          Buje_Final := L2B1
        barrenosTotales := 27
        barrenoActual := 1
        Loop While (checkContinuously=false) expression=barrenoActual≤barrenosTotales
          MoveL speed 250 mm/s, acceleration 1200 mm/s^2 (useActiveTCP=true) feature=Base
            bajada_broca := p[0,0,0.009,0,0,0]
            internos := interpolate_pose(Buje_Inicial, Buje_Final, ((barrenoActual)-1)/((barrenosTotales)-1))
            Folder Alturas
              If barrenoActual≟3 or barrenoActual≟5 or barrenoActual≟7 or barrenoActual≟9 or barrenoActual≟11 or barrenoActual≟13 or barrenoActual≟15 or barrenoActual≟17 or barrenoActual≟19 or barrenoActual≟21 or barrenoActual≟23 or barrenoActual≟25 or barrenoActual≟27 or barrenoActual≟1
                Set ExpressionOutput pin=mensaje_mw10; expression=200
                Wait DigitalInput pin=Continuar_M30; digitalValue=1
                Wait Sleep waitTime=1
                Set ExpressionOutput pin=mensaje_mw10; expression=150
                Wait Sleep waitTime=1
              MoveJ speed 60 deg/s, acceleration 80 deg/s^2 (useActiveTCP=true) feature=Base
                Waypoint Waypoint (Variable): variable=internos
              Wait Sleep waitTime=2
              If P1h[2]<P2h[2]
                acomodin := (altura/(barrenosTotales-1))*(barrenoActual-1)
                tcp_chido := get_actual_tcp_pose()
                offset_bajada := p[tcp_chido[0],tcp_chido[1],((alta-0.0095)-(acomodin/1000)),tcp_chido[3],tcp_chido[4],tcp_chido[5]]
                MoveL speed 15 mm/s, acceleration 30 mm/s^2 (useActiveTCP=true) feature=Base
                  Waypoint Waypoint (Variable): variable=offset_bajada
              Else 
                acomodin := (altura/(barrenosTotales-1))*(26-(barrenoActual-1))
                tcp_chido := get_actual_tcp_pose()
                offset_bajada := p[tcp_chido[0],tcp_chido[1],((alta-0.0095)-(acomodin/1000)),tcp_chido[3],tcp_chido[4],tcp_chido[5]]
                MoveL speed 15 mm/s, acceleration 30 mm/s^2 (useActiveTCP=true) feature=Base
                  Waypoint Waypoint (Variable): variable=offset_bajada
            Folder Freemove
              Wait Sleep waitTime=2
              Script: freedrive_mode()
              Wait Sleep waitTime=2.5
              Script: end_freedrive_mode()
            Wait Sleep waitTime=0.3
            Set DigitalOutput pin=config_out[1]; digitalValue=1
            Wait Sleep waitTime=1
            Wait Sleep waitTime=0.3
            Wait Sleep waitTime=0.3
            Wait Sleep waitTime=0.3
            Loop Counting (count=2) loopVariable(name=Loop_74)
              Poses_taladrado := pose_sub(get_actual_tcp_pose(), bajada_broca)
              Waypoint Waypoint (Variable): motionParameters(jointSpeed=1.047198 jointAcceleration=1.396263 cartesianSpeed=0.001 cartesianAcceleration=0.005); variable=Poses_taladrado
              If bajada_broca≟p[0,0,0.018,0,0,0]
                num_barreno := str_cat("Barreno: ",barrenoActual)
                tcp_actual := get_actual_tcp_pose()
                X_actual := str_cat("     X: ",tcp_actual[0])
                Y_actual := str_cat("     Y: ",tcp_actual[1])
                pos_barreno := str_cat(X_actual,Y_actual)
                Script: textmsg(num_barreno,pos_barreno)
              Poses_taladrado := pose_add(get_actual_tcp_pose(), bajada_broca)
              Waypoint Waypoint (Variable): motionParameters(jointSpeed=1.047198 jointAcceleration=1.396263 cartesianSpeed=0.01 cartesianAcceleration=0.01); variable=Poses_taladrado
              bajada_broca := pose_add(bajada_broca, p[0,0,0.009,0,0,0])
            MoveDirectionNode (selectedDirection=ZPlus toolParams=0.03, 0.04)
              Until DISTANCE (allowActions=false deceleration=3 distanceNodeType=STOP) Distance=0.05; motionParameters(blendRadius=0)
            MoveJ speed 60 deg/s, acceleration 80 deg/s^2 (useActiveTCP=true) feature=Base
              Waypoint Waypoint (Variable): variable=internos
            Wait Sleep waitTime=0.3
            Set DigitalOutput pin=config_out[1]; digitalValue=0
            Wait Sleep waitTime=0.3
            If barrenoActual≟13
              MoveDirectionNode (selectedDirection=ZPlus)
                Until DISTANCE (allowActions=false deceleration=3 distanceNodeType=STOP) Distance=0.03; motionParameters(blendRadius=0)
              MoveJ speed 60 deg/s, acceleration 80 deg/s^2 (useActiveTCP=true) feature=Base
                Waypoint Zona_izq1: TCP in base x=721.637 y=-174.262 z=505.425 mm, rx=2.3235 ry=2.1144 rz=0.0001 rad; joints [0.067, -89.734, -90.405, -179.332, -89.71, -0.034] deg
                Waypoint Posicion_Cero: TCP in base x=0.551 y=-324.742 z=1651.532 mm, rx=-0.0041 ry=-0.0154 rz=-3.05 rad; joints [-0.003, -90.003, 0.004, -89.999, -0.001, 0] deg
              Call Quitar_Broca_Chida
              Call Poner_Broca
              MoveJ speed 60 deg/s, acceleration 80 deg/s^2 (useActiveTCP=true) feature=Base
                Waypoint Posicion_Cero: TCP in base x=0.551 y=-324.742 z=1651.532 mm, rx=-0.0041 ry=-0.0154 rz=-3.05 rad; joints [-0.003, -90.003, 0.004, -89.999, -0.001, 0] deg
                Waypoint Zona_izq1: TCP in base x=721.637 y=-174.262 z=505.425 mm, rx=2.3235 ry=2.1144 rz=0.0001 rad; joints [0.067, -89.734, -90.405, -179.332, -89.71, -0.034] deg
            ElseIf barrenoActual≟27
              MoveDirectionNode (selectedDirection=ZPlus)
                Until DISTANCE (allowActions=false deceleration=3 distanceNodeType=STOP) Distance=0.03; motionParameters(blendRadius=0)
              MoveJ speed 60 deg/s, acceleration 80 deg/s^2 (useActiveTCP=true) feature=Base
                Waypoint Zona_izq1: TCP in base x=721.637 y=-174.262 z=505.425 mm, rx=2.3235 ry=2.1144 rz=0.0001 rad; joints [0.067, -89.734, -90.405, -179.332, -89.71, -0.034] deg
                Waypoint Posicion_Cero: TCP in base x=0.551 y=-324.742 z=1651.532 mm, rx=-0.0041 ry=-0.0154 rz=-3.05 rad; joints [-0.003, -90.003, 0.004, -89.999, -0.001, 0] deg
              Call Quitar_Broca_Chida
              Set DigitalOutput pin=carrusel_home; digitalValue=1
              Wait Sleep waitTime=1
              Set DigitalOutput pin=carrusel_home; digitalValue=0
              Set ExpressionOutput pin=mensaje_mw10; expression=85
              Wait DigitalInput pin=Continuar_M30; digitalValue=1
              Wait Sleep waitTime=1
              Set ExpressionOutput pin=mensaje_mw10; expression=120
              Wait DigitalInput pin=Continuar_M30; digitalValue=1
              Wait Sleep waitTime=1
              Set DigitalOutput pin=carrusel_home; digitalValue=1
              Wait Sleep waitTime=1
              Set DigitalOutput pin=carrusel_home; digitalValue=0
              Set ExpressionOutput pin=mensaje_mw10; expression=90
              Wait DigitalInput pin=Continuar_M30; digitalValue=1
              Wait Sleep waitTime=1
              Call Poner_Broca
              broca := 217
              MoveJ speed 60 deg/s, acceleration 80 deg/s^2 (useActiveTCP=true) feature=Base
                Waypoint Posicion_Cero: TCP in base x=0.551 y=-324.742 z=1651.532 mm, rx=-0.0041 ry=-0.0154 rz=-3.05 rad; joints [-0.003, -90.003, 0.004, -89.999, -0.001, 0] deg
                Waypoint Zona_izq1: TCP in base x=721.637 y=-174.262 z=505.425 mm, rx=2.3235 ry=2.1144 rz=0.0001 rad; joints [0.067, -89.734, -90.405, -179.332, -89.71, -0.034] deg
              Set ExpressionOutput pin=mensaje_mw10; expression=95
              Wait DigitalInput pin=Continuar_M30; digitalValue=1
              Wait Sleep waitTime=1
              Set ExpressionOutput pin=mensaje_mw10; expression=150
              Wait DigitalInput pin=Continuar_M30; digitalValue=1
              Wait Sleep waitTime=1
            barrenoActual := barrenoActual+1
      Folder Linea 1 a 217
        broca := 217
        Folder Buje_inicial
          Buje_Inicial := L1B2
        Folder Buje_final
          Buje_Final := L1B1
        barrenosTotales := 27
        barrenoActual := 1
        Loop While (checkContinuously=false) expression=barrenoActual≤barrenosTotales
          MoveL speed 250 mm/s, acceleration 1200 mm/s^2 (useActiveTCP=true) feature=Base
            bajada_broca := p[0,0,0.018,0,0,0]
            internos := interpolate_pose(Buje_Inicial, Buje_Final, ((barrenoActual)-1)/((barrenosTotales)-1))
            Folder Alturas
              If barrenoActual≟3 or barrenoActual≟5 or barrenoActual≟7 or barrenoActual≟9 or barrenoActual≟11 or barrenoActual≟13 or barrenoActual≟15 or barrenoActual≟17 or barrenoActual≟19 or barrenoActual≟21 or barrenoActual≟23 or barrenoActual≟25 or barrenoActual≟27 or barrenoActual≟1
                Set ExpressionOutput pin=mensaje_mw10; expression=200
                Wait DigitalInput pin=Continuar_M30; digitalValue=1
                Wait Sleep waitTime=1
                Set ExpressionOutput pin=mensaje_mw10; expression=150
                Wait Sleep waitTime=1
              MoveJ speed 60 deg/s, acceleration 80 deg/s^2 (useActiveTCP=true) feature=Base
                Waypoint Waypoint (Variable): variable=internos
              Wait Sleep waitTime=2
              If P1h[2]<P2h[2]
                acomodin := (altura/(barrenosTotales-1))*(barrenoActual-1)
                tcp_chido := get_actual_tcp_pose()
                offset_bajada := p[tcp_chido[0],tcp_chido[1],((alta-0.0095)-(acomodin/1000)),tcp_chido[3],tcp_chido[4],tcp_chido[5]]
                MoveL speed 15 mm/s, acceleration 30 mm/s^2 (useActiveTCP=true) feature=Base
                  Waypoint Waypoint (Variable): variable=offset_bajada
              Else 
                acomodin := (altura/(barrenosTotales-1))*(26-(barrenoActual-1))
                tcp_chido := get_actual_tcp_pose()
                offset_bajada := p[tcp_chido[0],tcp_chido[1],((alta-0.0095)-(acomodin/1000)),tcp_chido[3],tcp_chido[4],tcp_chido[5]]
                MoveL speed 15 mm/s, acceleration 30 mm/s^2 (useActiveTCP=true) feature=Base
                  Waypoint Waypoint (Variable): variable=offset_bajada
            Folder Freemove
              Wait Sleep waitTime=2
              Script: freedrive_mode()
              Wait Sleep waitTime=2.5
              Script: end_freedrive_mode()
            Wait Sleep waitTime=0.3
            Set DigitalOutput pin=config_out[1]; digitalValue=1
            Wait Sleep waitTime=1
            Wait Sleep waitTime=0.3
            Wait Sleep waitTime=0.3
            Wait Sleep waitTime=0.3
            Loop Counting (count=1) loopVariable(name=Loop_76)
              Poses_taladrado := pose_sub(get_actual_tcp_pose(), bajada_broca)
              Waypoint Waypoint (Variable): motionParameters(jointSpeed=1.047198 jointAcceleration=1.396263 cartesianSpeed=0.001 cartesianAcceleration=0.005); variable=Poses_taladrado
              If bajada_broca≟p[0,0,0.018,0,0,0]
